// TwinCAT 3 PLC project Building_1_5_Totes_ARUP
// ProgramVersion: 3.1.4023.0
// libraries:
//   Tc2_Standard, * (Beckhoff Automation GmbH)
//   Tc2_System, * (Beckhoff Automation GmbH)
//   Tc2_TcpIp, * (Beckhoff Automation GmbH)
//   Tc2_Utilities, * (Beckhoff Automation GmbH)
//   Tc3_Module, * (Beckhoff Automation GmbH)
// project tree:
//   DUTs/EAP/ E_EAP_PubType.TcDUT, ST_EAP_DEVICE.TcDUT, ST_EAP_Publisher.TcDUT, ST_EAP_Pub_Variable.TcDUT, ST_EAP_Subscriber.TcDUT, ST_EAP_Sub_Variable.TcDUT
//   DUTs/ E_EquipType.TcTLEO, E_StatusCode.TcDUT, ST_EquipmentStatus.TcDUT, ST_SafetyState.TcDUT
//   DUTs/Messages/ E_EquipmentUpdate.TcTLEO, E_MessageIds.TcTLEO, E_TransportComplete.TcDUT, E_TransportResponse.TcTLEO, ST_Msg_ConveyorStat.TcDUT, ST_Msg_EquipStat.TcDUT
//   FunctionBlocks/BarCode/ CognexDataMan260.TcPOU
//   FunctionBlocks/Binder/ BinderX_ReleaseControl.TcPOU, FB_BinderPusher.TcPOU, FB_Binder_SingulateHold.TcPOU
//   FunctionBlocks/Binder/DUTs/ ST_Binder.TcDUT, ST_BinderState.TcDUT, ST_FromBinder.TcDUT, ST_ToBinder.TcDUT
//   FunctionBlocks/Conveyance/DUTs/ E_ConvType.TcDUT
//   FunctionBlocks/Conveyance/ FB_CnvyrCnfig_1.TcPOU, FB_SleepCntrl.TcPOU
//   FunctionBlocks/Divert/DUTs/ ST_Divert.TcDUT, ST_DivertCfg.TcDUT
//   FunctionBlocks/Divert/Functions/ FB_ConfirmCheck.TcPOU, FB_DivertCommission.TcPOU, FB_DivertControl.TcPOU, FB_DivertDecision.TcPOU, FB_DivertFullMonitor.TcPOU, FB_DivertLog.TcPOU
//   FunctionBlocks/Encoder/DUTs/ ST_Encoder.TcDUT
//   FunctionBlocks/Encoder/ FB_ProcessEncoder.TcPOU
//   FunctionBlocks/FB_Merge/ E_MergeState.TcDUT, FB_Merge2.TcPOU, MergeExample.TcPOU, ST_MergeSts.TcDUT
//   FunctionBlocks/FB_Merge/Merge Inlet/ FB_MergeInlet.TcPOU, ST_MergeInlet.TcDUT, ST_MergeInletCfg.TcDUT, ST_MergeInletCtrl.TcDUT, ST_MergeInletSts.TcDUT
//   FunctionBlocks/FB_MotionMerge/ FB_MotionMerge.TcPOU, MotionMergeExample.TcPOU, ST_MotionMergeConfig.TcDUT, ST_MotionMergeItem.TcDUT
//   FunctionBlocks/Item/DUTs/ ST_Item.TcDUT, ST_ItemBuffer.TcDUT, ST_ItemBufferFdbk.TcDUT, ST_ItemLogBuffer.TcDUT, ST_ItemTemporary.TcDUT
//   FunctionBlocks/Item/ FB_ItemBuffer.TcPOU, FB_ItemLogBuffer.TcPOU
//   FunctionBlocks/LEDControl/ FB_LEDModeCtrl.TcPOU, ST_HMILEDMode.TcDUT, ST_LEDMode.TcDUT, ST_RGB.TcDUT
//   FunctionBlocks/Logging/ FB_UpdateLog.TcPOU, ST_LogMsg.TcDUT
//   FunctionBlocks/Metrics/ FB_Metrics.TcPOU
//   FunctionBlocks/Server/Data types/ E_ConnectionSteps.TcDUT, E_ServerSteps.TcDUT
//   FunctionBlocks/Server/ FB_Server.TcPOU, FB_ServerApplication.TcPOU, FB_ServerConnection.TcPOU
//   FunctionBlocks/Server/Helper POUs/ FB_FrameFifo.TcPOU, FB_LogFifo.TcPOU
//   FunctionBlocks/Singulation/ FB_Singulation.TcPOU, FB_TwoGripIndexer.TcPOU, FB_TwoGripSingulation.TcPOU
//   FunctionBlocks/Solenoids/Functions/ FB_Solenoid_DA.TcPOU, FB_Solenoid_SA.TcPOU
//   FunctionBlocks/Sorter/DUTs/ ST_RoundRobin.TcDUT, ST_RoundRobinCfg.TcDUT, ST_RoundRobinDest.TcDUT, ST_Sorter.TcDUT, ST_SorterConfig.TcDUT
//   FunctionBlocks/Sorter/Functions/ FB_FindDestination.TcPOU, FB_SorterLog.TcPOU
//   FunctionBlocks/Sorter/ ProcessBuffers.TcPOU, SorterExample.TcPOU, SorterProgram.TcPOU
//   FunctionBlocks/Sorter/VISUs/ ArrayInspection.TcVIS, DiverterTest.TcVIS, SorterArray.TcVIS
//   FunctionBlocks/StateControl/ E_OperStateCntrl.TcTLEO, E_StateCntrl.TcTLEO, E_StopCodes.TcTLEO, FB_ManageCodes.TcPOU, FB_StateCntrl.TcPOU, ST_StateCntrlPB.TcDUT, ST_StateCntrlSts.TcDUT
//   FunctionBlocks/Utils/Events/ FB_EventMngr.TcPOU, FB_Intlks_Latch.TcPOU, FB_Intlks_NoLatch.TcPOU, ST_CfgEvents.TcDUT, ST_EventSts.TcDUT
//   FunctionBlocks/Utils/ FB_AlrtStrtDelay.TcPOU, FB_EquipCntrl.TcPOU, FB_Flasher.TcPOU, FB_FlipFlop.TcPOU, FB_JamDetect.TcPOU, FB_PhotoEye.TcPOU, FB_SystemCntrl.TcPOU, F_CalculateDifference.TcPOU, F_CalculateIndex.TcPOU, F_DecIndex.TcPOU, F_IncIndex.TcPOU, F_PaddNumber.TcPOU, IncIndex.TcPOU, SystemCntrl_Example.TcPOU
//   FunctionBlocks/Utils/Filters/ FB_DigDebnce.TcPOU, FB_DigDebnce_Off.TcPOU, FB_DigDebnce_On.TcPOU, F_Clip.TcPOU
//   FunctionBlocks/VFD/DUTs/ DRIVE_STATE.TcTLEO
//   FunctionBlocks/VFD/Functions/ DriveState.TcPOU, VFD.TcPOU
//   / GlobalTextList.TcGTLO, PlcTask.TcTTO, Visualization Manager.TcVMO (not stored)
//   GVLs/ GVL_EquipArrays.TcGVL, GVL_IO.TcGVL, GVL_Logging.TcGVL, GVL_SorterItems.TcGVL
//   POUs/ BarCodeReaders.TcPOU, CommStatus.TcPOU, Conveyors.TcPOU, Log_Diverts_P2140.TcPOU, Log_Diverts_P2150.TcPOU, MAIN.TcPOU, MsgControl.TcPOU, Photoeyes.TcPOU, ProcessBuffers_P2150.TcPOU, ProcessBuffers_P2140.TcPOU, ProxSensors.TcPOU, P_PulseCountDist.TcPOU, ServerControl.TcPOU, Singulation_Control.TcPOU, Solenoids.TcPOU, Sorter.TcPOU, Sorter_P2140.TcPOU, Sorter_P2150.TcPOU, System.TcPOU, SystemSafety.TcPOU
// real-time tasks:
//   TASK PlcTask: cycle T#10ms, priority 20, ADS port 350
//   TASK BCR_Sync: cycle T#1ms, priority 1, ADS port 301
// I/O:
//   DEVICE Device 1 (EtherCAT), AmsNetId 5.84.5.4.2.1
//     Term 1 (EK1200) [EK1200-5000 EtherCAT Power supply (2A E-Bus)]
//       Term 2 (EL6070-0033)
//       PLC-7021 (EL1008) [EL1008 8Ch. Dig. Input 24V, 3ms]
//       PLC-8051 (EL2008) [EL2008 8Ch. Dig. Output 24V, 0.5A]
//       PLC-8431 (EL1918) [EL1918, 8Ch. Safety Input 24V, TwinSAFE]
//         modules: Module 2 (FSLOGIC)
//       PLC-9031 (EL5152) [EL5152 2Ch. Inc. Encoder]
//       PLC-10081 (EK1122) [EK1122 2 port EtherCAT junction] // RIOs
//         SRIO-1151 (EP1908) [EP1908, 8 Ch. Safety Input 24V, TwinSAFE ]
//           modules: Module 1 (FSOE)
//         RIO-2151 (EP2339-0022) [EP2339-0022 16 Ch. Dig. Input/Output 24V, 0,5A, M12]
//         RIO-3171 (EP2339-0022) [EP2339-0022 16 Ch. Dig. Input/Output 24V, 0,5A, M12]
//         RIO-4141 (EP2339-0022) [EP2339-0022 16 Ch. Dig. Input/Output 24V, 0,5A, M12]
//         SRIO-7151 (EP1908) [EP1908, 8 Ch. Safety Input 24V, TwinSAFE ]
//           modules: Module 1 (FSOE)
//         RIO-8171 (EP2339-0022) [EP2339-0022 16 Ch. Dig. Input/Output 24V, 0,5A, M12]
//         RIO-9191 (EP2339-0022) [EP2339-0022 16 Ch. Dig. Input/Output 24V, 0,5A, M12]
//         RIO-10161 (EP2339-0022) [EP2339-0022 16 Ch. Dig. Input/Output 24V, 0,5A, M12]
//         RIO-11171 (EP2339-0022) [EP2339-0022 16 Ch. Dig. Input/Output 24V, 0,5A, M12]
//         RIO12182 (EP2339-0022) [EP2339-0022 16 Ch. Dig. Input/Output 24V, 0,5A, M12]
//       PLC-10261 (EK1122) [EK1122 2 port EtherCAT junction] // MCC
//         Term 19 (EK1100) [EK1100 EtherCAT Coupler (2A E-Bus)]
//           PLC-12031 (EL2008) [EL2008 8Ch. Dig. Output 24V, 0.5A]
//           PLC-12221 (EL2008) [EL2008 8Ch. Dig. Output 24V, 0.5A]
//           PLC-12451 (EL1008) [EL1008 8Ch. Dig. Input 24V, 3ms]
//           PLC-12631 (EL1008) [EL1008 8Ch. Dig. Input 24V, 3ms]
//           PLC-13071 (EL2008) [EL2008 8Ch. Dig. Output 24V, 0.5A]
//           PLC-13471 (EL1008) [EL1008 8Ch. Dig. Input 24V, 3ms]
//           PLC-14061 (EL1918) [EL1918, 8Ch. Safety Input 24V, TwinSAFE]
//             modules: Module 1 (FSOE), Module 2 (FSLOGIC)
//           PLC-14461 (EL2904) [EL2904, 4 Ch. Safety Output 24V, 0.5A, TwinSAFE]
//             modules: Module 1 (FSOES), Module 2 (DO)
//           PLC-15101 (EK1122) [EK1122 2 port EtherCAT junction]
//             P2141 (Inverter i550 Cabinet) [i550 Cabinet V05.04.xx]
//             P2146 (Inverter i550 Cabinet) [i550 Cabinet V06.02.xx]
//             P3080 (Inverter i550 Cabinet) [i550 Cabinet V06.02.xx]
//   DEVICE Device 2 (RT-Ethernet Protocol), AmsNetId 5.84.5.4.3.1
//   DEVICE Communition with 205 (EtherCAT Automation Protocol), AmsNetId 5.84.5.4.4.1
//     Pub_To_205 (Publisher)
//     Sub_To_205 (Subscriber)
//   DEVICE Device 4 (TC3 EIP Scanner), AmsNetId 5.84.5.2.5.1
//     BCR_S2140_01 // <INFO> </INFO> <EDS> C:\TwinCAT\3.1\Config\Io\EtherNetIP\0678077313070100.eds </EDS>
//     BCR_S2141_2 // <INFO> </INFO> <EDS> C:\TwinCAT\3.1\Config\Io\EtherNetIP\0678077313070100.eds </EDS>
//     BCR_S2150_2 // <INFO> </INFO> <EDS> C:\TwinCAT\3.1\Config\Io\EtherNetIP\0678077313070100.eds </EDS>
//     BCR_S3080_01 // <INFO> </INFO> <EDS> C:\TwinCAT\3.1\Config\Io\EtherNetIP\0678077313070100.eds </EDS>
// variable links:
//   (this object) <-> Device 1 (EtherCAT)/Term 1 (EK1200)/PLC-10081 (EK1122)/SRIO-1151 (EP1908)
//     Term 1 (EK1200)/PLC-8431 (EL1918)/ConnectionInputs/Message_26 TxPDO <-> Module 1 (FSOE)/FSOE Outputs/FSOE
//     Term 1 (EK1200)/PLC-8431 (EL1918)/ConnectionOutputs/Message_26 RxPDO <-> Module 1 (FSOE)/FSOE Inputs/FSOE
//   (this object) <-> Device 1 (EtherCAT)/Term 1 (EK1200)/PLC-10081 (EK1122)/SRIO-7151 (EP1908)
//     Term 1 (EK1200)/PLC-8431 (EL1918)/ConnectionInputs/Message_25 TxPDO <-> Module 1 (FSOE)/FSOE Outputs/FSOE
//     Term 1 (EK1200)/PLC-8431 (EL1918)/ConnectionOutputs/Message_25 RxPDO <-> Module 1 (FSOE)/FSOE Inputs/FSOE
//   (this object) <-> Device 1 (EtherCAT)/Term 1 (EK1200)/PLC-10261 (EK1122)/Term 19 (EK1100)/PLC-14061 (EL1918)
//     Term 1 (EK1200)/PLC-8431 (EL1918)/ConnectionInputs/Message_29 TxPDO <-> Module 1 (FSOE)/FSoE Outputs/FSOE
//     Term 1 (EK1200)/PLC-8431 (EL1918)/ConnectionOutputs/Message_29 RxPDO <-> Module 1 (FSOE)/FSoE Inputs/FSOE
//   (this object) <-> Device 1 (EtherCAT)/Term 1 (EK1200)/PLC-10261 (EK1122)/Term 19 (EK1100)/PLC-14461 (EL2904)
//     Term 1 (EK1200)/PLC-8431 (EL1918)/ConnectionInputs/Message_27 TxPDO <-> Module 1 (FSOES)/RxPDO/FSOE
//     Term 1 (EK1200)/PLC-8431 (EL1918)/ConnectionOutputs/Message_27 RxPDO <-> Module 1 (FSOES)/TxPDO/FSOE
//   (this object) <-> Device 1 (EtherCAT)/Term 1 (EK1200)/PLC-8431 (EL1918)
//     Term 1 (EK1200)/PLC-10081 (EK1122)/SRIO-1151 (EP1908)/Module 1 (FSOE)/FSOE Inputs/FSOE <-> ConnectionOutputs/Message_26 RxPDO
//     Term 1 (EK1200)/PLC-10081 (EK1122)/SRIO-7151 (EP1908)/Module 1 (FSOE)/FSOE Inputs/FSOE <-> ConnectionOutputs/Message_25 RxPDO
//     Term 1 (EK1200)/PLC-10081 (EK1122)/SRIO-1151 (EP1908)/Module 1 (FSOE)/FSOE Outputs/FSOE <-> ConnectionInputs/Message_26 TxPDO
//     Term 1 (EK1200)/PLC-10081 (EK1122)/SRIO-7151 (EP1908)/Module 1 (FSOE)/FSOE Outputs/FSOE <-> ConnectionInputs/Message_25 TxPDO
//     Term 1 (EK1200)/PLC-10261 (EK1122)/Term 19 (EK1100)/PLC-14061 (EL1918)/Module 1 (FSOE)/FSoE Inputs/FSOE <-> ConnectionOutputs/Message_29 RxPDO
//     Term 1 (EK1200)/PLC-10261 (EK1122)/Term 19 (EK1100)/PLC-14061 (EL1918)/Module 1 (FSOE)/FSoE Outputs/FSOE <-> ConnectionInputs/Message_29 TxPDO
//     Term 1 (EK1200)/PLC-10261 (EK1122)/Term 19 (EK1100)/PLC-14461 (EL2904)/Module 1 (FSOES)/RxPDO/FSOE <-> ConnectionInputs/Message_27 TxPDO
//     Term 1 (EK1200)/PLC-10261 (EK1122)/Term 19 (EK1100)/PLC-14461 (EL2904)/Module 1 (FSOES)/TxPDO/FSOE <-> ConnectionOutputs/Message_27 RxPDO
//   Building_1_5_Totes_ARUP Instance <-> Communition with 205 (EtherCAT Automation Protocol)
//     PlcTask Inputs/MAIN.EAP_205.DevState <-> Inputs/DevState
//     PlcTask Outputs/MAIN.EAP_205.DevCtrl <-> Outputs/DevCtrl
//   Building_1_5_Totes_ARUP Instance <-> Communition with 205 (EtherCAT Automation Protocol)/Pub_To_205 (Publisher)
//     PlcTask Inputs/MAIN.EAP_205.Publisher.FrameState <-> Inputs/FrameState
//     PlcTask Inputs/MAIN.EAP_205.Publisher.Variables[0].VarState <-> To205_P2130_IsRunning/Inputs/VarState
//     PlcTask Inputs/MAIN.EAP_205.Publisher.Variables[1].VarState <-> To205_P3095_SendingProduct/Inputs/VarState
//     PlcTask Outputs/GVL_IO.To205_P2130_IsRunning <-> To205_P2130_IsRunning/Outputs/VarData
//     PlcTask Outputs/GVL_IO.To205_P3095_SendingProduct <-> To205_P3095_SendingProduct/Outputs/VarData
//     PlcTask Outputs/MAIN.EAP_205.Publisher.FrameCtrl <-> Outputs/FrameCtrl
//     PlcTask Outputs/MAIN.EAP_205.Publisher.IPAddr <-> Outputs/IpAddr
//     PlcTask Outputs/MAIN.EAP_205.Publisher.Variables[0].VarCtrl <-> To205_P2130_IsRunning/Outputs/VarCtrl
//     PlcTask Outputs/MAIN.EAP_205.Publisher.Variables[0].VarID <-> To205_P2130_IsRunning/Outputs/VarId
//     PlcTask Outputs/MAIN.EAP_205.Publisher.Variables[1].VarCtrl <-> To205_P3095_SendingProduct/Outputs/VarCtrl
//     PlcTask Outputs/MAIN.EAP_205.Publisher.Variables[1].VarID <-> To205_P3095_SendingProduct/Outputs/VarId
//   Building_1_5_Totes_ARUP Instance <-> Communition with 205 (EtherCAT Automation Protocol)/Sub_To_205 (Subscriber)
//     PlcTask Inputs/GVL_IO.From205_P2125_SendingProduct <-> From205_P2125_SendingProduct/Inputs/VarData
//     PlcTask Inputs/GVL_IO.From205_P3100_IsRunning <-> From205_P3100_IsRunning/Inputs/VarData
//     PlcTask Inputs/MAIN.EAP_205.Subscriber.FrameState <-> Inputs/FrameState
//     PlcTask Inputs/MAIN.EAP_205.Subscriber.Variables[0].CycleIndex <-> From205_P3100_IsRunning/Inputs/CycleIndex
//     PlcTask Inputs/MAIN.EAP_205.Subscriber.Variables[0].Quality <-> From205_P3100_IsRunning/Inputs/Quality
//     PlcTask Inputs/MAIN.EAP_205.Subscriber.Variables[0].VarState <-> From205_P3100_IsRunning/Inputs/VarState
//     PlcTask Inputs/MAIN.EAP_205.Subscriber.Variables[1].CycleIndex <-> From205_P2125_SendingProduct/Inputs/CycleIndex
//     PlcTask Inputs/MAIN.EAP_205.Subscriber.Variables[1].Quality <-> From205_P2125_SendingProduct/Inputs/Quality
//     PlcTask Inputs/MAIN.EAP_205.Subscriber.Variables[1].VarState <-> From205_P2125_SendingProduct/Inputs/VarState
//     PlcTask Outputs/MAIN.EAP_205.Subscriber.FrameCtrl <-> Outputs/FrameCtrl
//     PlcTask Outputs/MAIN.EAP_205.Subscriber.Variables[0].VarCtrl <-> From205_P3100_IsRunning/Outputs/VarCtrl
//     PlcTask Outputs/MAIN.EAP_205.Subscriber.Variables[0].VarId <-> From205_P3100_IsRunning/Outputs/VarId
//     PlcTask Outputs/MAIN.EAP_205.Subscriber.Variables[1].VarCtrl <-> From205_P2125_SendingProduct/Outputs/VarCtrl
//     PlcTask Outputs/MAIN.EAP_205.Subscriber.Variables[1].VarId <-> From205_P2125_SendingProduct/Outputs/VarId
//   Building_1_5_Totes_ARUP Instance <-> Device 1 (EtherCAT)/Term 1 (EK1200)/PLC-10081 (EK1122)/RIO-10161 (EP2339-0022)
//     PlcTask Inputs/GVL_IO.DS_P2135 <-> Channel 8/P2135 Motor Disconnect
//     PlcTask Inputs/GVL_IO.DS_P2140 <-> Channel 2/P2140 Motor Disconnect
//     PlcTask Inputs/GVL_IO.PB_RemoteReset_10221 <-> Channel 6/PB-10221
//     PlcTask Inputs/Photoeyes.PE_10081.In_PE <-> Channel 9/PE-10081
//     PlcTask Inputs/Photoeyes.PE_10091.In_PE <-> Channel 1/PE-10091
//     PlcTask Inputs/Photoeyes.PE_10151.In_PE <-> Channel 11/PE-10151
//     PlcTask Inputs/Photoeyes.PE_10291.In_PE <-> Channel 7/PE-10291
//     PlcTask Inputs/Photoeyes.PE_10302.In_PE <-> Channel 15/PE-10302
//     PlcTask Inputs/ProxSensors.In_PX_10181_Extended <-> Channel 12/PX-10181
//     PlcTask Inputs/ProxSensors.In_PX_10211_Extended <-> Channel 13/PX-10211
//     PlcTask Inputs/ProxSensors.In_PX_10231_Retracted <-> Channel 14/PX-10231
//     PlcTask Outputs/GVL_IO.LT_10161_Red <-> Channel 19/LT-10161
//     PlcTask Outputs/GVL_IO.LT_10171_Yellow <-> Channel 20/LT-10171
//     PlcTask Outputs/GVL_IO.LT_10201_Green <-> Channel 21/LT-10201
//     PlcTask Outputs/GVL_IO.PL2140_01_Extend <-> Channel 26/SV-10121
//   Building_1_5_Totes_ARUP Instance <-> Device 1 (EtherCAT)/Term 1 (EK1200)/PLC-10081 (EK1122)/RIO-11171 (EP2339-0022)
//     PlcTask Inputs/GVL_IO.RIO11171_WcState <-> WcState/WcState
//     PlcTask Inputs/Photoeyes.PE_11191.In_PE <-> Channel 11/PE-11191
//     PlcTask Inputs/Photoeyes.PE_11221.In_PE <-> Channel 12/PE11221
//     PlcTask Inputs/Photoeyes.PE_11241.In_PE <-> Channel 13/????PE11421
//     PlcTask Inputs/ProxSensors.In_PX_11141_Extended <-> Channel 9/PX-11141
//     PlcTask Inputs/ProxSensors.In_PX_11181_Extended <-> Channel 3/PX-11181
//     PlcTask Inputs/ProxSensors.In_PX_11291_Extended <-> Channel 7/PX-11291
//     PlcTask Inputs/ProxSensors.In_PX_11161_Retracted <-> Channel 10/PX-11161
//     PlcTask Inputs/ProxSensors.In_PX_11201_Retracted <-> Channel 4/PX-11201
//     PlcTask Inputs/ProxSensors.In_PX_11321_Retracted <-> Channel 8/PX-11321
//     PlcTask Outputs/GVL_IO.GR2140_01_Extend <-> Channel 22/SV-11261
//     PlcTask Outputs/GVL_IO.GR2140_02_Extend <-> Channel 21/SV-11241
//     PlcTask Outputs/GVL_IO.PI2140_01_Extend <-> Channel 17/SV-11121
//     PlcTask Outputs/GVL_IO.PI2140_01_Retract <-> Channel 18/SV-11151
//   Building_1_5_Totes_ARUP Instance <-> Device 1 (EtherCAT)/Term 1 (EK1200)/PLC-10081 (EK1122)/RIO-2151 (EP2339-0022)
//     PlcTask Inputs/GVL_IO.DS_P2145 <-> Channel 15/P2145 Motor Disconnect
//     PlcTask Inputs/GVL_IO.DS_P2146 <-> Channel 12/P2146 Motor Disconnect
//     PlcTask Inputs/GVL_IO.RIO2151_WcState <-> WcState/WcState
//     PlcTask Inputs/Photoeyes.PE_2101.In_PE <-> Channel 9/PE-2101
//     PlcTask Inputs/Photoeyes.PE_2131.In_PE <-> Channel 11/PE-2131
//     PlcTask Inputs/Photoeyes.PE_2201.In_PE <-> Channel 13/PE-2201
//     PlcTask Inputs/Photoeyes.PE_2231.In_PE <-> Channel 14/PE-2231
//     PlcTask Inputs/Photoeyes.PE_2301.In_PE <-> Channel 7/PE-2301
//     PlcTask Inputs/Photoeyes.PE_2331.In_PE <-> Channel 8/PE-2331
//     PlcTask Inputs/ProxSensors.In_PX_2131_Extended <-> Channel 1/PX-2131
//     PlcTask Inputs/ProxSensors.In_PX_2181_Extended <-> Channel 3/PX-2181
//     PlcTask Inputs/ProxSensors.In_PX_2151_Retracted <-> Channel 2/PX-2151
//     PlcTask Inputs/ProxSensors.In_PX_2201_Retracted <-> Channel 4/PX-2201
//     PlcTask Outputs/GVL_IO.GR2150_01_Extend <-> Channel 22/SV-2261
//     PlcTask Outputs/GVL_IO.PI2150_01_Extend <-> Channel 21/SV-2241
//   Building_1_5_Totes_ARUP Instance <-> Device 1 (EtherCAT)/Term 1 (EK1200)/PLC-10081 (EK1122)/RIO-3171 (EP2339-0022)
//     PlcTask Inputs/GVL_IO.PB_RemoteReset_3211 <-> Channel 12/PB-3211
//     PlcTask Inputs/GVL_IO.RIO3171_WcState <-> WcState/WcState
//     PlcTask Inputs/Photoeyes.PE_3111.In_PE <-> Channel 1/PE-3111
//     PlcTask Inputs/Photoeyes.PE_3231.In_PE <-> Channel 5/PE-3231
//     PlcTask Inputs/ProxSensors.In_PX_3171_Extended <-> Channel 3/PX-3171
//     PlcTask Inputs/ProxSensors.In_PX_3301_Extended <-> Channel 7/PX-3301
//     PlcTask Inputs/ProxSensors.In_PX_3191_Retracted <-> Channel 4/PX-3191
//     PlcTask Inputs/ProxSensors.In_PX_3331_Retracted <-> Channel 8/PX-3331
//     PlcTask Outputs/GVL_IO.LT_3131_Red <-> Channel 25/LT-3131
//     PlcTask Outputs/GVL_IO.LT_3151_Yellow <-> Channel 26/LT-3151
//     PlcTask Outputs/GVL_IO.LT_3201_Green <-> Channel 27/LT-3201
//     PlcTask Outputs/GVL_IO.PU2150_01_Extend <-> Channel 22/SV-3261
//     PlcTask Outputs/GVL_IO.PU2150_02_Extend <-> Channel 18/SV-3141
//   Building_1_5_Totes_ARUP Instance <-> Device 1 (EtherCAT)/Term 1 (EK1200)/PLC-10081 (EK1122)/RIO-4141 (EP2339-0022)
//     PlcTask Inputs/GVL_IO.DS_P2150 <-> Channel 9/P2150 Motor Discconnect
//     PlcTask Inputs/GVL_IO.RIO4141_WcState <-> WcState/WcState
//     PlcTask Inputs/Photoeyes.PE_4091.In_PE <-> Channel 1/PE-4091
//     PlcTask Inputs/Photoeyes.PE_4161.In_PE <-> Channel 11/PE-4161
//     PlcTask Inputs/Photoeyes.PE_4201.In_PE <-> Channel 5/PE-4201
//     PlcTask Inputs/ProxSensors.In_PX_4151_Extended <-> Channel 3/PX-4151
//     PlcTask Inputs/ProxSensors.In_PX_4291_Extended <-> Channel 7/PX-4291
//     PlcTask Inputs/ProxSensors.In_PX_4171_Retracted <-> Channel 4/PX-4171
//     PlcTask Inputs/ProxSensors.In_PX_4311_Retracted <-> Channel 8/PX-4311
//     PlcTask Outputs/GVL_IO.PU2150_03_Extend <-> Channel 22/SV-4241
//     PlcTask Outputs/GVL_IO.PU2150_04_Extend <-> Channel 18/SV-4121
//   Building_1_5_Totes_ARUP Instance <-> Device 1 (EtherCAT)/Term 1 (EK1200)/PLC-10081 (EK1122)/RIO-8171 (EP2339-0022)
//     PlcTask Inputs/GVL_IO.DS_P2141 <-> Channel 7/P2141 Motor Disconnect
//     PlcTask Inputs/GVL_IO.DS_P2142 <-> Channel 1/P2142 Motor Disconnect
//     PlcTask Inputs/GVL_IO.DS_P2143 <-> Channel 8/P2143 Motor Disconnect
//     PlcTask Inputs/GVL_IO.PB_RemoteReset_8251 <-> Channel 6/PB-8251
//     PlcTask Inputs/GVL_IO.RIO8171_WcState <-> WcState/WcState
//     PlcTask Inputs/Photoeyes.PE_8131.In_PE <-> Channel 9/PE-8131
//     PlcTask Inputs/Photoeyes.PE_8141.In_PE <-> Channel 2/PE-8141
//     PlcTask Inputs/Photoeyes.PE_8161.In_PE <-> Channel 10/PE-8161
//     PlcTask Outputs/GVL_IO.LT_8181_Red <-> Channel 19/LT-8181
//     PlcTask Outputs/GVL_IO.LT_8191_Yellow <-> Channel 20/LT-8191
//     PlcTask Outputs/GVL_IO.LT_8231_Green <-> Channel 21/LT-8231
//   Building_1_5_Totes_ARUP Instance <-> Device 1 (EtherCAT)/Term 1 (EK1200)/PLC-10081 (EK1122)/RIO-9191 (EP2339-0022)
//     PlcTask Inputs/GVL_IO.DS_P3080 <-> Channel 5/P3080 Motor Disconnect
//     PlcTask Inputs/GVL_IO.RIO9191_WcState <-> WcState/WcState
//     PlcTask Inputs/Photoeyes.PE_9141.In_PE <-> Channel 1/PE-9141
//     PlcTask Inputs/Photoeyes.PE_9161.In_PE <-> Channel 2/PE-9161
//     PlcTask Inputs/Photoeyes.PE_9191.In_PE <-> Channel 3/PE-9191
//     PlcTask Inputs/Photoeyes.PE_9221.In_PE <-> Channel 4/PE-9221
//   Building_1_5_Totes_ARUP Instance <-> Device 1 (EtherCAT)/Term 1 (EK1200)/PLC-10081 (EK1122)/RIO12182 (EP2339-0022)
//     PlcTask Inputs/GVL_IO.DS_P2130 <-> Channel 4/P2130 Motor Disconnect
//     PlcTask Inputs/GVL_IO.DS_P3085 <-> Channel 2/P3085 Motor Disconnect
//     PlcTask Inputs/GVL_IO.DS_P3090 <-> Channel 6/P3090 Motor Disconnect
//     PlcTask Inputs/GVL_IO.DS_P3095 <-> Channel 12/P3095 Motor Disconnect
//     PlcTask Inputs/GVL_IO.RIO12182_WcState <-> WcState/WcState
//     PlcTask Inputs/Photoeyes.PE_12091.In_PE <-> Channel 1/PE-12091
//     PlcTask Inputs/Photoeyes.PE_12121.In_PE <-> Channel 9/PE-12121
//     PlcTask Inputs/Photoeyes.PE_12171.In_PE <-> Channel 3/PE-12171
//     PlcTask Inputs/Photoeyes.PE_12181.In_PE <-> Channel 11/PE-12181
//     PlcTask Inputs/Photoeyes.PE_12271.In_PE <-> Channel 5/PE-12271
//     PlcTask Inputs/ProxSensors.In_PX_12151_Extended <-> Channel 10/PX-12151
//     PlcTask Inputs/ProxSensors.In_PX_12251_Extended <-> Channel 13/PX-12251
//   Building_1_5_Totes_ARUP Instance <-> Device 1 (EtherCAT)/Term 1 (EK1200)/PLC-10081 (EK1122)/SRIO-1151 (EP1908)
//     PlcTask Inputs/GVL_IO.RIO1151_WcState <-> WcState/WcState
//   Building_1_5_Totes_ARUP Instance <-> Device 1 (EtherCAT)/Term 1 (EK1200)/PLC-10081 (EK1122)/SRIO-7151 (EP1908)
//     PlcTask Inputs/GVL_IO.RIO7151_WcState <-> WcState/WcState
//   Building_1_5_Totes_ARUP Instance <-> Device 1 (EtherCAT)/Term 1 (EK1200)/PLC-10261 (EK1122)/Term 19 (EK1100)/PLC-12031 (EL2008)
//     PlcTask Outputs/GVL_IO.P2130_RUN <-> Channel 1/P2130 Run
//     PlcTask Outputs/GVL_IO.P2135_RUN <-> Channel 2/P2135 Run
//     PlcTask Outputs/GVL_IO.P2140_RUN <-> Channel 3/P2140 Run
//     PlcTask Outputs/GVL_IO.P2142_RUN <-> Channel 4/P2142 Run
//     PlcTask Outputs/GVL_IO.P2143_RUN <-> Channel 5/P2143 Run
//     PlcTask Outputs/GVL_IO.P2145_RUN <-> Channel 6/P2145 Run
//     PlcTask Outputs/GVL_IO.P2150_RUN <-> Channel 7/P2150 Run
//     PlcTask Outputs/GVL_IO.P3085_RUN <-> Channel 8/P3085 Run
//   Building_1_5_Totes_ARUP Instance <-> Device 1 (EtherCAT)/Term 1 (EK1200)/PLC-10261 (EK1122)/Term 19 (EK1100)/PLC-12221 (EL2008)
//     PlcTask Outputs/GVL_IO.P3090_RUN <-> Channel 1/P3090 Run
//     PlcTask Outputs/GVL_IO.P3095_RUN <-> Channel 2/P3095 Run
//   Building_1_5_Totes_ARUP Instance <-> Device 1 (EtherCAT)/Term 1 (EK1200)/PLC-10261 (EK1122)/Term 19 (EK1100)/PLC-12451 (EL1008)
//     PlcTask Inputs/GVL_IO.P2130_Faulted <-> Channel 1/P2130 Faulted
//     PlcTask Inputs/GVL_IO.P2135_Faulted <-> Channel 2/P2135 Faulted
//     PlcTask Inputs/GVL_IO.P2140_Faulted <-> Channel 3/P2140 Faulted
//     PlcTask Inputs/GVL_IO.P2142_Faulted <-> Channel 4/P2142 Faulted
//     PlcTask Inputs/GVL_IO.P2143_Faulted <-> Channel 5/P2143 Faulted
//     PlcTask Inputs/GVL_IO.P2145_Faulted <-> Channel 6/P2145 Faulted
//     PlcTask Inputs/GVL_IO.P2150_Faulted <-> Channel 7/P2150 Faulted
//     PlcTask Inputs/GVL_IO.P3085_Faulted <-> Channel 8/P3085 Faulted
//   Building_1_5_Totes_ARUP Instance <-> Device 1 (EtherCAT)/Term 1 (EK1200)/PLC-10261 (EK1122)/Term 19 (EK1100)/PLC-12631 (EL1008)
//     PlcTask Inputs/GVL_IO.P3090_Faulted <-> Channel 1/P3090 Faulted
//     PlcTask Inputs/GVL_IO.P3095_Faulted <-> Channel 2/P3095 Faulted
//   Building_1_5_Totes_ARUP Instance <-> Device 1 (EtherCAT)/Term 1 (EK1200)/PLC-10261 (EK1122)/Term 19 (EK1100)/PLC-15101 (EK1122)/P2141 (Inverter i550 Cabinet)
//     PlcTask Inputs/Conveyors.P2141_VFD.ActualVelocity <-> TPDO (A) Velocity/Actual speed
//     PlcTask Inputs/Conveyors.P2141_VFD.StatusWord <-> TPDO (A) Velocity/CiA status word
//     PlcTask Outputs/Conveyors.P2141_VFD.ControlWord <-> RPDO (A) Velocity/CiA control word
//     PlcTask Outputs/Conveyors.P2141_VFD.TargetVelocity <-> RPDO (A) Velocity/Set speed
//   Building_1_5_Totes_ARUP Instance <-> Device 1 (EtherCAT)/Term 1 (EK1200)/PLC-10261 (EK1122)/Term 19 (EK1100)/PLC-15101 (EK1122)/P2146 (Inverter i550 Cabinet)
//     PlcTask Inputs/Conveyors.P2146_VFD.ActualVelocity <-> TPDO (A) Velocity/Actual speed
//     PlcTask Inputs/Conveyors.P2146_VFD.StatusWord <-> TPDO (A) Velocity/CiA status word
//     PlcTask Outputs/Conveyors.P2146_VFD.ControlWord <-> RPDO (A) Velocity/CiA control word
//     PlcTask Outputs/Conveyors.P2146_VFD.TargetVelocity <-> RPDO (A) Velocity/Set speed
//   Building_1_5_Totes_ARUP Instance <-> Device 1 (EtherCAT)/Term 1 (EK1200)/PLC-10261 (EK1122)/Term 19 (EK1100)/PLC-15101 (EK1122)/P3080 (Inverter i550 Cabinet)
//     PlcTask Inputs/Conveyors.P3080_VFD.ActualVelocity <-> TPDO (A) Velocity/Actual speed
//     PlcTask Inputs/Conveyors.P3080_VFD.StatusWord <-> TPDO (A) Velocity/CiA status word
//     PlcTask Outputs/Conveyors.P3080_VFD.ControlWord <-> RPDO (A) Velocity/CiA control word
//     PlcTask Outputs/Conveyors.P3080_VFD.TargetVelocity <-> RPDO (A) Velocity/Set speed
//   Building_1_5_Totes_ARUP Instance <-> Device 1 (EtherCAT)/Term 1 (EK1200)/PLC-7021 (EL1008)
//     PlcTask Inputs/GVL_IO.PB_SysReset <-> Channel 3/PB-7061
//     PlcTask Inputs/GVL_IO.PB_SysStart <-> Channel 1/PB-7021
//     PlcTask Inputs/GVL_IO.PB_SysStop <-> Channel 2/PB-7041
//   Building_1_5_Totes_ARUP Instance <-> Device 1 (EtherCAT)/Term 1 (EK1200)/PLC-8051 (EL2008)
//     PlcTask Outputs/GVL_IO.HornMainPanel <-> Channel 1/AH-8051
//     PlcTask Outputs/GVL_IO.LT_MainPanelStack_Green <-> Channel 4/LT-8111
//     PlcTask Outputs/GVL_IO.LT_MainPanelStack_Red <-> Channel 2/LT-8071
//     PlcTask Outputs/GVL_IO.LT_MainPanelStack_Yellow <-> Channel 3/LT-8091
//   Building_1_5_Totes_ARUP Instance <-> Device 1 (EtherCAT)/Term 1 (EK1200)/PLC-8431 (EL1918)
//     PlcTask Inputs/GVL_IO.Remote_PullCord2142_OK <-> StandardInputs/Standard Out Var 10
//     PlcTask Inputs/GVL_IO.Remote_PullCord2150_OK <-> StandardInputs/Standard Out Var 28
//     PlcTask Inputs/SystemSafety.Safety_PanelEstop <-> StandardInputs/Standard Out Var 9
//     PlcTask Inputs/SystemSafety.Safety_SystemEstopsOK <-> StandardInputs/Standard Out Var 15
//     PlcTask Inputs/SystemSafety.System_SafetyState.ComErr <-> StandardInputs/Standard Out Var 16
//     PlcTask Inputs/SystemSafety.System_SafetyState.FBErr <-> StandardInputs/Standard Out Var 17
//     PlcTask Inputs/SystemSafety.System_SafetyState.InRun <-> StandardInputs/Standard Out Var 30
//     PlcTask Inputs/SystemSafety.System_SafetyState.OtherErr <-> StandardInputs/Standard Out Var 18
//     PlcTask Outputs/SystemSafety.System_SafetyState.CommErrAck <-> StandardOutputs/Standard In Var 31
//     PlcTask Outputs/SystemSafety.System_SafetyState.ErrAck <-> StandardOutputs/Standard In Var 1
//     PlcTask Outputs/SystemSafety.System_SafetyState.Reset <-> StandardOutputs/Standard In Var 5
//     PlcTask Outputs/SystemSafety.System_SafetyState.Run <-> StandardOutputs/Standard In Var 2
//   Building_1_5_Totes_ARUP Instance <-> Device 1 (EtherCAT)/Term 1 (EK1200)/PLC-9031 (EL5152)
//     PlcTask Inputs/GVL_IO.ENC_9031_Period <-> ENC Period Channel 2/Period value
//     PlcTask Inputs/GVL_IO.ENC_9091_Period <-> ENC Period Channel 1/Period value
//     PlcTask Inputs/GVL_IO.ENC_9031_Raw <-> ENC Status compact Channel 2/Counter value
//     PlcTask Inputs/GVL_IO.ENC_9091_Raw <-> ENC Status compact Channel 1/Counter value
//   Building_1_5_Totes_ARUP Instance <-> Device 2 (RT-Ethernet Protocol)
//     PlcTask Inputs/GVL_IO.EthernetAdapter_State <-> Inputs/DevState
//   Building_1_5_Totes_ARUP Instance <-> Device 4 (TC3 EIP Scanner)/BCR_S2140_01
//     PlcTask Inputs/BarCodeReaders.BCR_S2140_01.Acquiring <-> Connection 1 (Input/Output)/Inputs/Acquiring
//     PlcTask Inputs/BarCodeReaders.BCR_S2140_01.DecodeComplete <-> Connection 1 (Input/Output)/Inputs/Decode Complete
//     PlcTask Inputs/BarCodeReaders.BCR_S2140_01.Decoding <-> Connection 1 (Input/Output)/Inputs/Decoding
//     PlcTask Inputs/BarCodeReaders.BCR_S2140_01.DeviceState <-> Inputs/State
//     PlcTask Inputs/BarCodeReaders.BCR_S2140_01.ResultCode <-> Connection 1 (Input/Output)/Inputs/Result Code
//     PlcTask Inputs/BarCodeReaders.BCR_S2140_01.ResultData <-> Connection 1 (Input/Output)/Inputs/Result Data
//     PlcTask Inputs/BarCodeReaders.BCR_S2140_01.ResultData @bit 8 <-> Connection 1 (Input/Output)/Inputs/Result Data_1
//     PlcTask Inputs/BarCodeReaders.BCR_S2140_01.ResultData @bit 80 <-> Connection 1 (Input/Output)/Inputs/Result Data_10
//     PlcTask Inputs/BarCodeReaders.BCR_S2140_01.ResultData @bit 88 <-> Connection 1 (Input/Output)/Inputs/Result Data_11
//     PlcTask Inputs/BarCodeReaders.BCR_S2140_01.ResultData @bit 96 <-> Connection 1 (Input/Output)/Inputs/Result Data_12
//     PlcTask Inputs/BarCodeReaders.BCR_S2140_01.ResultData @bit 104 <-> Connection 1 (Input/Output)/Inputs/Result Data_13
//     PlcTask Inputs/BarCodeReaders.BCR_S2140_01.ResultData @bit 112 <-> Connection 1 (Input/Output)/Inputs/Result Data_14
//     PlcTask Inputs/BarCodeReaders.BCR_S2140_01.ResultData @bit 120 <-> Connection 1 (Input/Output)/Inputs/Result Data_15
//     PlcTask Inputs/BarCodeReaders.BCR_S2140_01.ResultData @bit 128 <-> Connection 1 (Input/Output)/Inputs/Result Data_16
//     PlcTask Inputs/BarCodeReaders.BCR_S2140_01.ResultData @bit 136 <-> Connection 1 (Input/Output)/Inputs/Result Data_17
//     PlcTask Inputs/BarCodeReaders.BCR_S2140_01.ResultData @bit 144 <-> Connection 1 (Input/Output)/Inputs/Result Data_18
//     PlcTask Inputs/BarCodeReaders.BCR_S2140_01.ResultData @bit 152 <-> Connection 1 (Input/Output)/Inputs/Result Data_19
//     PlcTask Inputs/BarCodeReaders.BCR_S2140_01.ResultData @bit 16 <-> Connection 1 (Input/Output)/Inputs/Result Data_2
//     PlcTask Inputs/BarCodeReaders.BCR_S2140_01.ResultData @bit 160 <-> Connection 1 (Input/Output)/Inputs/Result Data_20
//     PlcTask Inputs/BarCodeReaders.BCR_S2140_01.ResultData @bit 168 <-> Connection 1 (Input/Output)/Inputs/Result Data_21
//     PlcTask Inputs/BarCodeReaders.BCR_S2140_01.ResultData @bit 176 <-> Connection 1 (Input/Output)/Inputs/Result Data_22
//     PlcTask Inputs/BarCodeReaders.BCR_S2140_01.ResultData @bit 184 <-> Connection 1 (Input/Output)/Inputs/Result Data_23
//     PlcTask Inputs/BarCodeReaders.BCR_S2140_01.ResultData @bit 192 <-> Connection 1 (Input/Output)/Inputs/Result Data_24
//     PlcTask Inputs/BarCodeReaders.BCR_S2140_01.ResultData @bit 200 <-> Connection 1 (Input/Output)/Inputs/Result Data_25
//     PlcTask Inputs/BarCodeReaders.BCR_S2140_01.ResultData @bit 24 <-> Connection 1 (Input/Output)/Inputs/Result Data_3
//     PlcTask Inputs/BarCodeReaders.BCR_S2140_01.ResultData @bit 32 <-> Connection 1 (Input/Output)/Inputs/Result Data_4
//     PlcTask Inputs/BarCodeReaders.BCR_S2140_01.ResultData @bit 40 <-> Connection 1 (Input/Output)/Inputs/Result Data_5
//     PlcTask Inputs/BarCodeReaders.BCR_S2140_01.ResultData @bit 48 <-> Connection 1 (Input/Output)/Inputs/Result Data_6
//     PlcTask Inputs/BarCodeReaders.BCR_S2140_01.ResultData @bit 56 <-> Connection 1 (Input/Output)/Inputs/Result Data_7
//     PlcTask Inputs/BarCodeReaders.BCR_S2140_01.ResultData @bit 64 <-> Connection 1 (Input/Output)/Inputs/Result Data_8
//     PlcTask Inputs/BarCodeReaders.BCR_S2140_01.ResultData @bit 72 <-> Connection 1 (Input/Output)/Inputs/Result Data_9
//     PlcTask Inputs/BarCodeReaders.BCR_S2140_01.ResultID <-> Connection 1 (Input/Output)/Inputs/Result ID
//     PlcTask Inputs/BarCodeReaders.BCR_S2140_01.ResultLength <-> Connection 1 (Input/Output)/Inputs/Result Length
//     PlcTask Inputs/BarCodeReaders.BCR_S2140_01.ResultsAvail <-> Connection 1 (Input/Output)/Inputs/Results Available
//     PlcTask Inputs/BarCodeReaders.BCR_S2140_01.TriggerAck <-> Connection 1 (Input/Output)/Inputs/Trigger Ack
//     PlcTask Inputs/BarCodeReaders.BCR_S2140_01.TriggerID <-> Connection 1 (Input/Output)/Inputs/Trigger ID
//     PlcTask Inputs/BarCodeReaders.BCR_S2140_01.TriggerReady <-> Connection 1 (Input/Output)/Inputs/Trigger Ready
//     PlcTask Outputs/BarCodeReaders.BCR_S2140_01.ResultsAck <-> Connection 1 (Input/Output)/Outputs/Results Ack
//     PlcTask Outputs/BarCodeReaders.BCR_S2140_01.Trigger <-> Connection 1 (Input/Output)/Outputs/Trigger
//     PlcTask Outputs/BarCodeReaders.BCR_S2140_01.TriggerEnable <-> Connection 1 (Input/Output)/Outputs/Trigger Enable
//   Building_1_5_Totes_ARUP Instance <-> Device 4 (TC3 EIP Scanner)/BCR_S2141_2
//     PlcTask Inputs/BarCodeReaders.BCR_S2141_01.Acquiring <-> Connection 2 (Input/Output)/Inputs/Acquiring
//     PlcTask Inputs/BarCodeReaders.BCR_S2141_01.DecodeComplete <-> Connection 2 (Input/Output)/Inputs/Decode Complete
//     PlcTask Inputs/BarCodeReaders.BCR_S2141_01.Decoding <-> Connection 2 (Input/Output)/Inputs/Decoding
//     PlcTask Inputs/BarCodeReaders.BCR_S2141_01.DeviceState <-> Inputs/State
//     PlcTask Inputs/BarCodeReaders.BCR_S2141_01.ResultCode <-> Connection 2 (Input/Output)/Inputs/Result Code
//     PlcTask Inputs/BarCodeReaders.BCR_S2141_01.ResultData <-> Connection 2 (Input/Output)/Inputs/Result Data
//     PlcTask Inputs/BarCodeReaders.BCR_S2141_01.ResultData @bit 8 <-> Connection 2 (Input/Output)/Inputs/Result Data_1
//     PlcTask Inputs/BarCodeReaders.BCR_S2141_01.ResultData @bit 80 <-> Connection 2 (Input/Output)/Inputs/Result Data_10
//     PlcTask Inputs/BarCodeReaders.BCR_S2141_01.ResultData @bit 88 <-> Connection 2 (Input/Output)/Inputs/Result Data_11
//     PlcTask Inputs/BarCodeReaders.BCR_S2141_01.ResultData @bit 96 <-> Connection 2 (Input/Output)/Inputs/Result Data_12
//     PlcTask Inputs/BarCodeReaders.BCR_S2141_01.ResultData @bit 104 <-> Connection 2 (Input/Output)/Inputs/Result Data_13
//     PlcTask Inputs/BarCodeReaders.BCR_S2141_01.ResultData @bit 112 <-> Connection 2 (Input/Output)/Inputs/Result Data_14
//     PlcTask Inputs/BarCodeReaders.BCR_S2141_01.ResultData @bit 120 <-> Connection 2 (Input/Output)/Inputs/Result Data_15
//     PlcTask Inputs/BarCodeReaders.BCR_S2141_01.ResultData @bit 128 <-> Connection 2 (Input/Output)/Inputs/Result Data_16
//     PlcTask Inputs/BarCodeReaders.BCR_S2141_01.ResultData @bit 136 <-> Connection 2 (Input/Output)/Inputs/Result Data_17
//     PlcTask Inputs/BarCodeReaders.BCR_S2141_01.ResultData @bit 144 <-> Connection 2 (Input/Output)/Inputs/Result Data_18
//     PlcTask Inputs/BarCodeReaders.BCR_S2141_01.ResultData @bit 152 <-> Connection 2 (Input/Output)/Inputs/Result Data_19
//     PlcTask Inputs/BarCodeReaders.BCR_S2141_01.ResultData @bit 16 <-> Connection 2 (Input/Output)/Inputs/Result Data_2
//     PlcTask Inputs/BarCodeReaders.BCR_S2141_01.ResultData @bit 160 <-> Connection 2 (Input/Output)/Inputs/Result Data_20
//     PlcTask Inputs/BarCodeReaders.BCR_S2141_01.ResultData @bit 168 <-> Connection 2 (Input/Output)/Inputs/Result Data_21
//     PlcTask Inputs/BarCodeReaders.BCR_S2141_01.ResultData @bit 176 <-> Connection 2 (Input/Output)/Inputs/Result Data_22
//     PlcTask Inputs/BarCodeReaders.BCR_S2141_01.ResultData @bit 184 <-> Connection 2 (Input/Output)/Inputs/Result Data_23
//     PlcTask Inputs/BarCodeReaders.BCR_S2141_01.ResultData @bit 192 <-> Connection 2 (Input/Output)/Inputs/Result Data_24
//     PlcTask Inputs/BarCodeReaders.BCR_S2141_01.ResultData @bit 200 <-> Connection 2 (Input/Output)/Inputs/Result Data_25
//     PlcTask Inputs/BarCodeReaders.BCR_S2141_01.ResultData @bit 24 <-> Connection 2 (Input/Output)/Inputs/Result Data_3
//     PlcTask Inputs/BarCodeReaders.BCR_S2141_01.ResultData @bit 32 <-> Connection 2 (Input/Output)/Inputs/Result Data_4
//     PlcTask Inputs/BarCodeReaders.BCR_S2141_01.ResultData @bit 40 <-> Connection 2 (Input/Output)/Inputs/Result Data_5
//     PlcTask Inputs/BarCodeReaders.BCR_S2141_01.ResultData @bit 48 <-> Connection 2 (Input/Output)/Inputs/Result Data_6
//     PlcTask Inputs/BarCodeReaders.BCR_S2141_01.ResultData @bit 56 <-> Connection 2 (Input/Output)/Inputs/Result Data_7
//     PlcTask Inputs/BarCodeReaders.BCR_S2141_01.ResultData @bit 64 <-> Connection 2 (Input/Output)/Inputs/Result Data_8
//     PlcTask Inputs/BarCodeReaders.BCR_S2141_01.ResultData @bit 72 <-> Connection 2 (Input/Output)/Inputs/Result Data_9
//     PlcTask Inputs/BarCodeReaders.BCR_S2141_01.ResultID <-> Connection 2 (Input/Output)/Inputs/Result ID
//     PlcTask Inputs/BarCodeReaders.BCR_S2141_01.ResultLength <-> Connection 2 (Input/Output)/Inputs/Result Length
//     PlcTask Inputs/BarCodeReaders.BCR_S2141_01.ResultsAvail <-> Connection 2 (Input/Output)/Inputs/Results Available
//     PlcTask Inputs/BarCodeReaders.BCR_S2141_01.TriggerAck <-> Connection 2 (Input/Output)/Inputs/Trigger Ack
//     PlcTask Inputs/BarCodeReaders.BCR_S2141_01.TriggerID <-> Connection 2 (Input/Output)/Inputs/Trigger ID
//     PlcTask Inputs/BarCodeReaders.BCR_S2141_01.TriggerReady <-> Connection 2 (Input/Output)/Inputs/Trigger Ready
//     PlcTask Outputs/BarCodeReaders.BCR_S2141_01.ResultsAck <-> Connection 2 (Input/Output)/Outputs/Results Ack
//     PlcTask Outputs/BarCodeReaders.BCR_S2141_01.Trigger <-> Connection 2 (Input/Output)/Outputs/Trigger
//     PlcTask Outputs/BarCodeReaders.BCR_S2141_01.TriggerEnable <-> Connection 2 (Input/Output)/Outputs/Trigger Enable
//   Building_1_5_Totes_ARUP Instance <-> Device 4 (TC3 EIP Scanner)/BCR_S2150_2
//     PlcTask Inputs/BarCodeReaders.BCR_S2150_01.Acquiring <-> Connection 2 (Input/Output)/Inputs/Acquiring
//     PlcTask Inputs/BarCodeReaders.BCR_S2150_01.DecodeComplete <-> Connection 2 (Input/Output)/Inputs/Decode Complete
//     PlcTask Inputs/BarCodeReaders.BCR_S2150_01.Decoding <-> Connection 2 (Input/Output)/Inputs/Decoding
//     PlcTask Inputs/BarCodeReaders.BCR_S2150_01.DeviceState <-> Inputs/State
//     PlcTask Inputs/BarCodeReaders.BCR_S2150_01.ResultCode <-> Connection 2 (Input/Output)/Inputs/Result Code
//     PlcTask Inputs/BarCodeReaders.BCR_S2150_01.ResultData <-> Connection 2 (Input/Output)/Inputs/Result Data
//     PlcTask Inputs/BarCodeReaders.BCR_S2150_01.ResultData @bit 8 <-> Connection 2 (Input/Output)/Inputs/Result Data_1
//     PlcTask Inputs/BarCodeReaders.BCR_S2150_01.ResultData @bit 80 <-> Connection 2 (Input/Output)/Inputs/Result Data_10
//     PlcTask Inputs/BarCodeReaders.BCR_S2150_01.ResultData @bit 88 <-> Connection 2 (Input/Output)/Inputs/Result Data_11
//     PlcTask Inputs/BarCodeReaders.BCR_S2150_01.ResultData @bit 96 <-> Connection 2 (Input/Output)/Inputs/Result Data_12
//     PlcTask Inputs/BarCodeReaders.BCR_S2150_01.ResultData @bit 104 <-> Connection 2 (Input/Output)/Inputs/Result Data_13
//     PlcTask Inputs/BarCodeReaders.BCR_S2150_01.ResultData @bit 112 <-> Connection 2 (Input/Output)/Inputs/Result Data_14
//     PlcTask Inputs/BarCodeReaders.BCR_S2150_01.ResultData @bit 120 <-> Connection 2 (Input/Output)/Inputs/Result Data_15
//     PlcTask Inputs/BarCodeReaders.BCR_S2150_01.ResultData @bit 128 <-> Connection 2 (Input/Output)/Inputs/Result Data_16
//     PlcTask Inputs/BarCodeReaders.BCR_S2150_01.ResultData @bit 136 <-> Connection 2 (Input/Output)/Inputs/Result Data_17
//     PlcTask Inputs/BarCodeReaders.BCR_S2150_01.ResultData @bit 144 <-> Connection 2 (Input/Output)/Inputs/Result Data_18
//     PlcTask Inputs/BarCodeReaders.BCR_S2150_01.ResultData @bit 152 <-> Connection 2 (Input/Output)/Inputs/Result Data_19
//     PlcTask Inputs/BarCodeReaders.BCR_S2150_01.ResultData @bit 16 <-> Connection 2 (Input/Output)/Inputs/Result Data_2
//     PlcTask Inputs/BarCodeReaders.BCR_S2150_01.ResultData @bit 160 <-> Connection 2 (Input/Output)/Inputs/Result Data_20
//     PlcTask Inputs/BarCodeReaders.BCR_S2150_01.ResultData @bit 168 <-> Connection 2 (Input/Output)/Inputs/Result Data_21
//     PlcTask Inputs/BarCodeReaders.BCR_S2150_01.ResultData @bit 176 <-> Connection 2 (Input/Output)/Inputs/Result Data_22
//     PlcTask Inputs/BarCodeReaders.BCR_S2150_01.ResultData @bit 184 <-> Connection 2 (Input/Output)/Inputs/Result Data_23
//     PlcTask Inputs/BarCodeReaders.BCR_S2150_01.ResultData @bit 192 <-> Connection 2 (Input/Output)/Inputs/Result Data_24
//     PlcTask Inputs/BarCodeReaders.BCR_S2150_01.ResultData @bit 200 <-> Connection 2 (Input/Output)/Inputs/Result Data_25
//     PlcTask Inputs/BarCodeReaders.BCR_S2150_01.ResultData @bit 24 <-> Connection 2 (Input/Output)/Inputs/Result Data_3
//     PlcTask Inputs/BarCodeReaders.BCR_S2150_01.ResultData @bit 32 <-> Connection 2 (Input/Output)/Inputs/Result Data_4
//     PlcTask Inputs/BarCodeReaders.BCR_S2150_01.ResultData @bit 40 <-> Connection 2 (Input/Output)/Inputs/Result Data_5
//     PlcTask Inputs/BarCodeReaders.BCR_S2150_01.ResultData @bit 48 <-> Connection 2 (Input/Output)/Inputs/Result Data_6
//     PlcTask Inputs/BarCodeReaders.BCR_S2150_01.ResultData @bit 56 <-> Connection 2 (Input/Output)/Inputs/Result Data_7
//     PlcTask Inputs/BarCodeReaders.BCR_S2150_01.ResultData @bit 64 <-> Connection 2 (Input/Output)/Inputs/Result Data_8
//     PlcTask Inputs/BarCodeReaders.BCR_S2150_01.ResultData @bit 72 <-> Connection 2 (Input/Output)/Inputs/Result Data_9
//     PlcTask Inputs/BarCodeReaders.BCR_S2150_01.ResultID <-> Connection 2 (Input/Output)/Inputs/Result ID
//     PlcTask Inputs/BarCodeReaders.BCR_S2150_01.ResultLength <-> Connection 2 (Input/Output)/Inputs/Result Length
//     PlcTask Inputs/BarCodeReaders.BCR_S2150_01.ResultsAvail <-> Connection 2 (Input/Output)/Inputs/Results Available
//     PlcTask Inputs/BarCodeReaders.BCR_S2150_01.TriggerAck <-> Connection 2 (Input/Output)/Inputs/Trigger Ack
//     PlcTask Inputs/BarCodeReaders.BCR_S2150_01.TriggerID <-> Connection 2 (Input/Output)/Inputs/Trigger ID
//     PlcTask Inputs/BarCodeReaders.BCR_S2150_01.TriggerReady <-> Connection 2 (Input/Output)/Inputs/Trigger Ready
//     PlcTask Outputs/BarCodeReaders.BCR_S2150_01.ResultsAck <-> Connection 2 (Input/Output)/Outputs/Results Ack
//     PlcTask Outputs/BarCodeReaders.BCR_S2150_01.Trigger <-> Connection 2 (Input/Output)/Outputs/Trigger
//     PlcTask Outputs/BarCodeReaders.BCR_S2150_01.TriggerEnable <-> Connection 2 (Input/Output)/Outputs/Trigger Enable
//   Building_1_5_Totes_ARUP Instance <-> Device 4 (TC3 EIP Scanner)/BCR_S3080_01
//     PlcTask Inputs/BarCodeReaders.BCR_S3080_01.Acquiring <-> Connection 2 (Input/Output)/Inputs/Acquiring
//     PlcTask Inputs/BarCodeReaders.BCR_S3080_01.DecodeComplete <-> Connection 2 (Input/Output)/Inputs/Decode Complete
//     PlcTask Inputs/BarCodeReaders.BCR_S3080_01.Decoding <-> Connection 2 (Input/Output)/Inputs/Decoding
//     PlcTask Inputs/BarCodeReaders.BCR_S3080_01.DeviceState <-> Inputs/State
//     PlcTask Inputs/BarCodeReaders.BCR_S3080_01.ResultCode <-> Connection 2 (Input/Output)/Inputs/Result Code
//     PlcTask Inputs/BarCodeReaders.BCR_S3080_01.ResultData <-> Connection 2 (Input/Output)/Inputs/Result Data
//     PlcTask Inputs/BarCodeReaders.BCR_S3080_01.ResultData @bit 8 <-> Connection 2 (Input/Output)/Inputs/Result Data_1
//     PlcTask Inputs/BarCodeReaders.BCR_S3080_01.ResultData @bit 80 <-> Connection 2 (Input/Output)/Inputs/Result Data_10
//     PlcTask Inputs/BarCodeReaders.BCR_S3080_01.ResultData @bit 88 <-> Connection 2 (Input/Output)/Inputs/Result Data_11
//     PlcTask Inputs/BarCodeReaders.BCR_S3080_01.ResultData @bit 96 <-> Connection 2 (Input/Output)/Inputs/Result Data_12
//     PlcTask Inputs/BarCodeReaders.BCR_S3080_01.ResultData @bit 104 <-> Connection 2 (Input/Output)/Inputs/Result Data_13
//     PlcTask Inputs/BarCodeReaders.BCR_S3080_01.ResultData @bit 112 <-> Connection 2 (Input/Output)/Inputs/Result Data_14
//     PlcTask Inputs/BarCodeReaders.BCR_S3080_01.ResultData @bit 120 <-> Connection 2 (Input/Output)/Inputs/Result Data_15
//     PlcTask Inputs/BarCodeReaders.BCR_S3080_01.ResultData @bit 128 <-> Connection 2 (Input/Output)/Inputs/Result Data_16
//     PlcTask Inputs/BarCodeReaders.BCR_S3080_01.ResultData @bit 136 <-> Connection 2 (Input/Output)/Inputs/Result Data_17
//     PlcTask Inputs/BarCodeReaders.BCR_S3080_01.ResultData @bit 144 <-> Connection 2 (Input/Output)/Inputs/Result Data_18
//     PlcTask Inputs/BarCodeReaders.BCR_S3080_01.ResultData @bit 152 <-> Connection 2 (Input/Output)/Inputs/Result Data_19
//     PlcTask Inputs/BarCodeReaders.BCR_S3080_01.ResultData @bit 16 <-> Connection 2 (Input/Output)/Inputs/Result Data_2
//     PlcTask Inputs/BarCodeReaders.BCR_S3080_01.ResultData @bit 160 <-> Connection 2 (Input/Output)/Inputs/Result Data_20
//     PlcTask Inputs/BarCodeReaders.BCR_S3080_01.ResultData @bit 168 <-> Connection 2 (Input/Output)/Inputs/Result Data_21
//     PlcTask Inputs/BarCodeReaders.BCR_S3080_01.ResultData @bit 176 <-> Connection 2 (Input/Output)/Inputs/Result Data_22
//     PlcTask Inputs/BarCodeReaders.BCR_S3080_01.ResultData @bit 184 <-> Connection 2 (Input/Output)/Inputs/Result Data_23
//     PlcTask Inputs/BarCodeReaders.BCR_S3080_01.ResultData @bit 192 <-> Connection 2 (Input/Output)/Inputs/Result Data_24
//     PlcTask Inputs/BarCodeReaders.BCR_S3080_01.ResultData @bit 200 <-> Connection 2 (Input/Output)/Inputs/Result Data_25
//     PlcTask Inputs/BarCodeReaders.BCR_S3080_01.ResultData @bit 24 <-> Connection 2 (Input/Output)/Inputs/Result Data_3
//     PlcTask Inputs/BarCodeReaders.BCR_S3080_01.ResultData @bit 32 <-> Connection 2 (Input/Output)/Inputs/Result Data_4
//     PlcTask Inputs/BarCodeReaders.BCR_S3080_01.ResultData @bit 40 <-> Connection 2 (Input/Output)/Inputs/Result Data_5
//     PlcTask Inputs/BarCodeReaders.BCR_S3080_01.ResultData @bit 48 <-> Connection 2 (Input/Output)/Inputs/Result Data_6
//     PlcTask Inputs/BarCodeReaders.BCR_S3080_01.ResultData @bit 56 <-> Connection 2 (Input/Output)/Inputs/Result Data_7
//     PlcTask Inputs/BarCodeReaders.BCR_S3080_01.ResultData @bit 64 <-> Connection 2 (Input/Output)/Inputs/Result Data_8
//     PlcTask Inputs/BarCodeReaders.BCR_S3080_01.ResultData @bit 72 <-> Connection 2 (Input/Output)/Inputs/Result Data_9
//     PlcTask Inputs/BarCodeReaders.BCR_S3080_01.ResultID <-> Connection 2 (Input/Output)/Inputs/Result ID
//     PlcTask Inputs/BarCodeReaders.BCR_S3080_01.ResultLength <-> Connection 2 (Input/Output)/Inputs/Result Length
//     PlcTask Inputs/BarCodeReaders.BCR_S3080_01.ResultsAvail <-> Connection 2 (Input/Output)/Inputs/Results Available
//     PlcTask Inputs/BarCodeReaders.BCR_S3080_01.TriggerAck <-> Connection 2 (Input/Output)/Inputs/Trigger Ack
//     PlcTask Inputs/BarCodeReaders.BCR_S3080_01.TriggerID <-> Connection 2 (Input/Output)/Inputs/Trigger ID
//     PlcTask Inputs/BarCodeReaders.BCR_S3080_01.TriggerReady <-> Connection 2 (Input/Output)/Inputs/Trigger Ready
//     PlcTask Outputs/BarCodeReaders.BCR_S3080_01.ResultsAck <-> Connection 2 (Input/Output)/Outputs/Results Ack
//     PlcTask Outputs/BarCodeReaders.BCR_S3080_01.Trigger <-> Connection 2 (Input/Output)/Outputs/Trigger
//     PlcTask Outputs/BarCodeReaders.BCR_S3080_01.TriggerEnable <-> Connection 2 (Input/Output)/Outputs/Trigger Enable

CONFIGURATION Building_1_5_Totes_ARUP
    RESOURCE PLC ON TwinCAT3
        TASK PlcTask(INTERVAL := T#10ms, PRIORITY := 20);
        PROGRAM MAIN WITH PlcTask : MAIN;
    END_RESOURCE
END_CONFIGURATION

// ---- DUTs/EAP/E_EAP_PubType.TcDUT
{attribute 'qualified_only'}
{attribute 'strict'}
TYPE E_EAP_PubType :
(
	e_AmsNetID 	:= 0,
	e_IPAddr	:= 1,
	e_MAC_ID	:= 2
);
END_TYPE

// ---- DUTs/EAP/ST_EAP_DEVICE.TcDUT
{attribute 'OPC.UA.DA' := '1'}
TYPE ST_EAP_DEVICE :
STRUCT
	DevName				:	STRING;		// Name of the EAP Device
	NetID				: 	STRING;		// Net ID of the EAP Device
	DevState	AT %I*	: 	UINT;		// EAP Device State
	DevCtrl		AT %Q*	: 	UINT;		// EAP Device Control
	Publisher			: 	ST_EAP_Publisher;		// Assumes single EAP to Publisher relationship
	Subscriber			: 	ST_EAP_Subscriber;		// Assumes single EAP to Subscriber relationship
END_STRUCT
END_TYPE

// ---- DUTs/EAP/ST_EAP_Publisher.TcDUT
TYPE ST_EAP_Publisher :
STRUCT
	Name				: 	STRING;		// Name of the EAP Publisher
	FrameState	AT %I*	: 	UINT;		// EAP FrameState, FrameState.0 = Not Transmitting, .1 = Frame too large, .2 = Subscriber Miissing
	FrameCtrl	AT %Q*	: 	UINT;		// EAP FrameCtrl, FrameCtrl.0 = Disable Sending, .1 = Remove destination MAC from ARP
	PubType				:	E_EAP_PubType := 0;	// EAP Publisher Type, AMS NetID (0), IP Address (1), MAC ID (2)
	NetID		AT %Q*	: 	AMSNETID;	// EAP Changeable NetID
	IPAddr		AT %Q*	: 	UDINT;		// EAP Changeable IP, stored as a single UDINT
	HMI_IPAddr			: 	USINTARR4;	// Used to enter IP Address on the HMI, MEMCPY function copies array to IPAddr 
	HMI_IPAddrDisp		: 	USINTARR4;	// Used to Display IP Address on the HMI, MEMCPY function copies IPAddr to Array 
	MACID		AT %Q*	: 	USINTARR6;	// EAP Changeable MAC ID, stored as an array of 6 USINT
	Variables			:	ARRAY[0..9] OF ST_EAP_Pub_Variable;		// Array of Published variables
END_STRUCT
END_TYPE

// ---- DUTs/EAP/ST_EAP_Pub_Variable.TcDUT
TYPE ST_EAP_Pub_Variable :
STRUCT
	Name				: 	STRING;		// Name of the Variable
	VarState	AT %I*	:	UINT;		// VarState.0 = Not Sent, 1 = Transmission Suspended, 0 = Transmission OK
	VarID 		AT %Q*	:	UINT;		// Changeable ID of the variable
	VarCtrl		AT %Q*	:	UINT;		// VarCtrl.0 = Disable publishing
END_STRUCT
END_TYPE

// ---- DUTs/EAP/ST_EAP_Subscriber.TcDUT
TYPE ST_EAP_Subscriber :
STRUCT
	Name				: 	STRING;		// Name of the EAP Subscriber
	FrameState	AT %I*	:	UINT;		// EAP FrameState, unused
	FrameCtrl	AT %Q*	:	UINT;		// EAP FrameCtrl, unused
	Variables			:	ARRAY[0..9] OF ST_EAP_Sub_Variable;		// Array of Subscribed variables
END_STRUCT
END_TYPE

// ---- DUTs/EAP/ST_EAP_Sub_Variable.TcDUT
TYPE ST_EAP_Sub_Variable :
STRUCT
	Name				: 	STRING;		// Name of the Variable
	VarState	AT %I*	:	UINT;		// VarState.0 = Invalid Hash/Version, .1 = Invalid Variable Length
	Quality		AT %I*	:	UINT;		// <>0, Duration the variable is not refreshed (in 100µs)
	CycleIndex	AT %I*	:	UINT;		// Incremented each publisher cycle
	VarId		AT %Q*	:	UINT;		// Changable Variable ID
	VarCtrl		AT %Q*	:	UINT;		// VarCtrl.1 = Ignore Hash/Version
END_STRUCT
END_TYPE

// ---- DUTs/E_EquipType.TcTLEO
{attribute 'qualified_only'}
{attribute 'strict'}
TYPE E_EquipType :
(
	Unknown := 0,
	System := 1,
	Conveyor := 2,
	Merge := 3,
	Gripper_SA := 4,
	Gripper_DA :=5,
	PinStop := 6,
	Pusher := 7,
	Divert := 8
) DINT;
END_TYPE

// ---- DUTs/E_StatusCode.TcDUT
{attribute 'qualified_only'}
{attribute 'strict'}
(*
	0-19 	-System level faults
	20-39	-Sorter Transfer Specific Status Codes
	40-59	-Diverter Transfer Specific Status Codes
	60-79	-Transfer Specific Status Codes
*)
TYPE E_StatusCode :
(
	No_Status				:= 0,
	OK						:= 1,
	Stopped					:= 2,
	Faulted					:= 3,	
	UnknownError	 		:= 9,	
	
	NotInSorter				:= 20,	
	UpdateRequested			:= 21,
	QueryNeeded				:= 22,
	UpdateNeeded 			:= 23,
	UpdateReceived 			:= 24,
	ReqNotReceived			:= 25,
	ItemNotUpdated			:= 26,
	UnidentifiedItem		:= 27,
	ItemNotFound			:= 28,
	Sorter_UnknownError 	:= 29,
	Assign_Accepted			:= 30,
	Assign_Full				:= 31,
	Assign_NotFound			:= 32,
	Assign_NotInducted		:= 33,
	Exiting_Sorter			:= 34,
	Exited_Sorter			:= 35,
	
	Divert_Idle				:= 40,
	In_Sorter 				:= 41,
	Diverting 				:= 42,
	Divert_Missed 			:= 43,
	Divert_Full				:= 44,
	Divert_Offline			:= 45,
	Divert_Faulted			:= 46,
	Divert_NotInducted		:= 47,
	Divert_LateAssignment	:= 48,
	Divert_UnknownError 	:= 49,
	Divert_Recirculated		:= 50,
	Divert_Detected			:= 51,
	Divert_Success			:= 52,
	Divert_Complete			:= 53,
	
	In_Transfer 			:= 61,
	Transferring 			:= 62,
	Tranfer_Success	 		:= 63,
	Transfer_Missed 		:= 64,
	Transfer_Failed 		:= 65,	
	Transfer_UnknownError 	:= 69
) USINT;
END_TYPE

// ---- DUTs/Messages/E_EquipmentUpdate.TcTLEO
{attribute 'qualified_only'}
{attribute 'strict'}
TYPE E_EquipmentUpdate :
(
	Manual := 1,
	Auto := 2,
	Offline := 3,
	Running := 4,
	SleepActive := 5,
	Faulted := 6,
	OverHeight := 7
);
END_TYPE

// ---- DUTs/Messages/E_MessageIds.TcTLEO
//{attribute 'qualified_only'}
{attribute 'strict'}
TYPE E_MessageIds :
(
	NoMessage_00 := 0,
	TransportCommand_05 := 5,
	LocationUpdateResponse_07 := 7,
	EquipmentStatusResponse_08 := 8,
	KeepAlive_09 := 9,
	Arrival_23 := 23,
	TransportResponse_25 := 25,
	TransportComplete_26 := 26,
	LocationUpdate_27 := 27,
	EquipmentStatusUpdate_28 := 28,
	KeepAliveResponse_29 := 29
);
END_TYPE

// ---- DUTs/Messages/E_TransportComplete.TcDUT
{attribute 'qualified_only'}
{attribute 'strict'}
TYPE E_TransportComplete :
(
	Success := 0,
	Unavailable := 1,
	Faulted := 2,
	Offline := 3,
	Passed := 8,
	ConfirmFailed := 11,
	InductFailed := 12
)INT ;
END_TYPE

// ---- DUTs/Messages/E_TransportResponse.TcTLEO
{attribute 'qualified_only'}
{attribute 'strict'}
TYPE E_TransportResponse :
(
	Accepted := 0,
	DivertLaneUnavailable := 1,
	LoadIdNotFound := 2,
	UnknownFailure := 11,
	NextLoadReady := 12,
	LateInduction := 13
);
END_TYPE

// ---- DUTs/Messages/ST_Msg_ConveyorStat.TcDUT
TYPE ST_Msg_ConveyorStat :
STRUCT
	DeviceID:	STRING(5);
	Status:	INT;
END_STRUCT
END_TYPE

// ---- DUTs/Messages/ST_Msg_EquipStat.TcDUT
TYPE ST_Msg_EquipStat :
STRUCT
	DeviceID:	STRING(5);
	Status:	INT;
END_STRUCT
END_TYPE

// ---- DUTs/ST_EquipmentStatus.TcDUT
TYPE ST_EquipmentStatus :
STRUCT
	Sts_EquipmentState:	ST_StateCntrlSts;		// State Status
	Sts_SleepingActive: BOOL;	// Status to show conveyor is in sleep state
	Sts_All_Intlks_OK:	BOOL;		// Status bit to show that all interloks are good to Run 
	Sts_FaultActive:	BOOL;	// Status Bit Showing that a fault is present (0= No Active Faults, 1= Fault Active)
	Sts_WarnActive:	BOOL;	// Status Bit Showing that a warning is present (0= No Active Warnings, 1= Warning Active)
	Sts_All_Evnts_OK: BOOL;		// Status Bit Showing that ALL Events are OK to RUN (0= Event Present, 1= OK to Run)
	Sts_IsRunning :BOOL;	// Status to show conveyor is running (1=running)
	Sts_IsExtending :BOOL;	// Status to show Actuator is extending (1=extending)
	Sts_IsExtended :BOOL;	// Status to show Actuator is extended (1=extended)
	Sts_IsRetracting :BOOL;	// Status to show Actuator is retracting (1=retracting)
	Sts_IsRetracted :BOOL;	// Status to show Actuator is retracted (1=retracted)
END_STRUCT
END_TYPE

// ---- DUTs/ST_SafetyState.TcDUT
TYPE ST_SafetyState :
STRUCT
	Reset 	 	AT %Q* : BOOL;
	Run 	 	AT %Q* : BOOL;
	ErrAck 	 	AT %Q* : BOOL;
	CommErrAck	AT %Q*	:BOOL;
	ComErr    	AT %I* : BOOL;
	FBErr     	AT %I* : BOOL;
	OtherErr  	AT %I* : BOOL;
	InRun 		AT %I* : BOOL;
END_STRUCT
END_TYPE

// ---- FunctionBlocks/Binder/DUTs/ST_Binder.TcDUT
{attribute 'OPC.UA.DA' := '1'}
TYPE ST_Binder :
STRUCT
	State		:	ST_BinderState;		// State of the Binder
	FromBinder	:	ST_FromBinder;		// Data Recevied from the Binder
	ToBinder	:	ST_ToBinder;		// Data Sent to the Binder
END_STRUCT
END_TYPE

// ---- FunctionBlocks/Binder/DUTs/ST_BinderState.TcDUT
TYPE ST_BinderState :
STRUCT
	DoorOpenOK  	AT %I*: BOOL;
	EstopOK  		AT %I*: BOOL;
	NetReset		AT %I*: BOOL;
	VlvBankPower 	AT %I*: BOOL;
	DumpValve 		AT %I*: BOOL;
	SystemEstopOK	AT %I*: BOOL;
END_STRUCT
END_TYPE

// ---- FunctionBlocks/Binder/DUTs/ST_FromBinder.TcDUT
TYPE ST_FromBinder :
STRUCT
	ProcessingComplete :BOOL;
	Online: BOOL;
	RackProcessing : BOOL;
END_STRUCT
END_TYPE

// ---- FunctionBlocks/Binder/DUTs/ST_ToBinder.TcDUT
TYPE ST_ToBinder :
STRUCT
	ProductHeld : BOOL;
	StatusSingulator : UINT;
END_STRUCT
END_TYPE

// ---- FunctionBlocks/Conveyance/DUTs/E_ConvType.TcDUT
{attribute 'qualified_only'}
{attribute 'strict'}
TYPE E_ConvType :
(
	standard 	:= 0,
	end			:= 1,
	slave		:= 2
);
END_TYPE

// ---- FunctionBlocks/Divert/DUTs/ST_Divert.TcDUT
{attribute 'OPC.UA.DA' := '1'}
TYPE ST_Divert :
STRUCT
	{attribute 'OPC.UA.DA' := '0'}
	Config			: ST_DivertCfg;		// Configuration Variables

	Full 			: BOOL;				//Diverter full photo eye is blocked
	Jammed 			: BOOL;				//Jammed photo eye is blocked
	Faulted 		: BOOL;				//Returned faulted status
	Available 		: BOOL;				//Return availability status, auto/running/etc.  Will depend on the system and requirements

	Status 			: E_StatusCode := E_StatusCode.Divert_Idle; 	//Status Code, initialized to Idle

	ConfirmPE	   	: BOOL;				//Physical input address of photo eye
	FullPE		   	: BOOL;				//Physical input address of photo eye
	JamPE		   	: BOOL;				//Physical input address of photo eye 
	Output1	 		: BOOL;				//Physical output address of diverter
	Output2	  		: BOOL;				//Physical output address of diverter
	
	{attribute 'OPC.UA.DA' := '0'}
	Output1Flag		: DINT;				//Indicates what the encoder count is when output is energized
	
	FullTime		: TIME;				//Time that full PE has to be high before the lane is considered full     
	{attribute 'OPC.UA.DA' := '0'}
	FullTimer		: TON; 				//Timer that is used for checking how long the full PE is on
	
	{attribute 'OPC.UA.DA' := '0'}
	Item			: ST_Item;			// Currently Diverting Item
END_STRUCT
END_TYPE

// ---- FunctionBlocks/Divert/DUTs/ST_DivertCfg.TcDUT
{attribute 'OPC.UA.DA' := '1'}
TYPE ST_DivertCfg :
STRUCT
	ID 				: STRING;			// User assigned Divert indetifier		
	EquipID 		: STRING[5];		// Identifier used for host communication		
	Number			: INT;				// Divert number, can be distinct from the Index in the Divert Array
	Distance		: INT;				// Distance, in encoder counts, from induct photo eye
	ConfirmDist		: INT;				// Distance from the Divert point to the Confirm PE
	Direction		: BOOL;				// 0 = Divert to one side, 1 = Divert to the other side 
	FullTime		: REAL;				// Time, in seconds, that full PE has to be high before the lane is considered full
	IsDischarge		: BOOL;				// TRUE, process and test for items destined for non-discharge diverts that missed
END_STRUCT
END_TYPE

// ---- FunctionBlocks/Encoder/DUTs/ST_Encoder.TcDUT
TYPE ST_Encoder :
STRUCT
	EncoderRawCount : UDINT;	// Raw encoder Count, acommodates 16 and 32 bit encoder resoultions
	CurrentCount : UDINT;		// Current Pulse Count
	BitMaskSize	: UINT;			// Number of bits to mask into the CurrentCount from the Actual Encoder Pulses
	EncoderString	: STRING;	// Encoder pulses formatted as string
END_STRUCT
END_TYPE

// ---- FunctionBlocks/FB_Merge/E_MergeState.TcDUT
{attribute 'qualified_only'}
//{attribute 'strict'}
TYPE E_MergeState :
(
	stStopped := 0,
	stClearTakeAway := 1,
	stMergeOperational := 2,
	stMergeManual := 3
)INT;
END_TYPE

// ---- FunctionBlocks/FB_Merge/Merge Inlet/ST_MergeInlet.TcDUT
{attribute 'OPC.UA.DA' := '1'}
TYPE ST_MergeInlet :
STRUCT
	{attribute 'OPC.UA.DA' := '0'}
	Cfg		:	ST_MergeInletCfg;
	Ctrl	:	ST_MergeInletCtrl;
END_STRUCT
END_TYPE

// ---- FunctionBlocks/FB_Merge/Merge Inlet/ST_MergeInletCfg.TcDUT
{attribute 'OPC.UA.DA' := '1'}
TYPE ST_MergeInletCfg :
STRUCT
	Cfg_UseMtrFdBck				:	BOOL := FALSE;	// Configuration bit to determine if motor feed back is used (1= use feedback)
	Cfg_UseHighWaterPE			:	BOOL := FALSE;	// Configuration bit to determine if the High Water indicator PE is used (1= use High Water PE)
	Cfg_UseHiHiWaterPE			:	BOOL := FALSE;	// Configuration bit to determine if the HiHi Water indicator PE is used (1= use HiHi Water PE)
	Cfg_HighTriggerTime			:	REAL := 1;		// Time that full trigger has to be on to record high condition
	Cfg_HiHiTriggerTime			:	REAL := 1;		// Time that full trigger has to be on to record hihi condition
	Cfg_HiHiClearTime			:	REAL := 10;		// Time Merge runs in response to a HiHi Water condition
	Cfg_MrgReqPrdctWaitTime		: 	REAL := 45;		// Time that product has to wait for full mark to be reached before requesting merge
	Cfg_ReleaseCount			:	INT := 1;		// Required count to be released before switching merge locations
	Cfg_ReleaseCountWaitTime	:	REAL := 60;		// Time to wait to achieve release count before switching merge locations
	Cfg_ClearRunOutTime			:	REAL := 25;		// Time to wait for product to clear the merge
	Cfg_MergeName				:	STRING(20);		// Name used to Identify the Merge on the HMI
END_STRUCT
END_TYPE

// ---- FunctionBlocks/FB_Merge/Merge Inlet/ST_MergeInletCtrl.TcDUT
{attribute 'OPC.UA.DA' := '1'}
TYPE ST_MergeInletCtrl :
STRUCT
	PhotoEyeDischarge			:	BOOL;			// Photo Eye at the discharge of the assigned merge location
	PhotoEyeEntryHigh			:	BOOL;			// Photo Eye at the Full (high water) location of the merge
	PhotoEyeEntryHiHi			:	BOOL;			// Photo Eye at the Full (hihi water) location of the merge
	MergeInletMtrFdBck			:	BOOL;			// Current motor feedback for the assigned merge location
	In_InletState				:	E_StateCntrl;	// The State of the merge take away conveyor
	In_oMergeRelease			:	BOOL;
	{attribute 'OPC.UA.DA' := '0'}
	SimActive					:	BOOL;			// Simulation Bit 
END_STRUCT
END_TYPE

// ---- FunctionBlocks/FB_Merge/Merge Inlet/ST_MergeInletSts.TcDUT
{attribute 'OPC.UA.DA' := '1'}
TYPE ST_MergeInletSts :
STRUCT
	MergeRequested				:	BOOL;		// Merge has been Requested (1=request Active)
	Granted						:	BOOL;		// The Granted state of this Inlet
	MergeComplete				:	BOOL;		// Flag to finish merging
	HiHiDetected				:	BOOL;		// HiHi Event has been detected and requires control
	HiHiTimedReleaseActive		:	BOOL;		// Indicates that a HiHi event clearout is in process
	Out_MergeInletRunActive		:	BOOL;		// Output for Merge inlet run
	Sts_MergeInletRun			:	BOOL;		// Merge Inlet status Motor is currently running (1=merging or running)
	MergeRunOutActive			:	BOOL;		// Flag to indicate that the Merge Run Out is active (1=active)
	CrrntReleaseCount			:	INT;		// The current count of product released
END_STRUCT
END_TYPE

// ---- FunctionBlocks/FB_Merge/ST_MergeSts.TcDUT
{attribute 'OPC.UA.DA' := '1'}
TYPE ST_MergeSts :
STRUCT
	MergeEnabled			: 	BOOL;		// Merge is enabled 
	MergeTakeAwayMtrActive	:	BOOL;		// Output for Merge take away motor
	MergeSubState			:	E_MergeState;
	MergeSubStateTxt		:	STRING(20);
	MergeJammed				:	BOOL;		// Merge is Jammed
	InletCount				:	INT;
END_STRUCT
END_TYPE

// ---- FunctionBlocks/FB_MotionMerge/ST_MotionMergeConfig.TcDUT
{attribute 'OPC.UA.DA' := '1'}
TYPE ST_MotionMergeConfig :
STRUCT
	MergeDistance: 			UINT;	// The distance from the induct PE to the merge point (Merge start location)
	MergeClearDistance: 	UINT;	// The distance from the induct PE to a cleared point past the merge (Merge end location)
	MergeOpening_Min: 		UINT;	// The minimum window size to allow a merge
	Item_ExtendFwd:			UINT;	// The distance to Extend the Item lead edge
	Item_ExtendRev:			UINT;	// The distance to Extend teh Item Trail edge
	MergeClearTime: 		REAL;	// The time, in seconds, to declare the merge clear
END_STRUCT
END_TYPE

// ---- FunctionBlocks/FB_MotionMerge/ST_MotionMergeItem.TcDUT
TYPE ST_MotionMergeItem :
STRUCT
	Count_InductStart	: UDINT;
	Count_InductEnd	: UDINT;
	Length	: UDINT;
	OnConveyor	: BOOL;
END_STRUCT
END_TYPE

// ---- FunctionBlocks/Item/DUTs/ST_Item.TcDUT
TYPE ST_Item :
STRUCT
	ID : STRING := '';		// Bar Code 	
	UniqueID : DINT := 0;		// Generic ID for tracking
	Destination : DINT := 0;
	DestinationIdx : DINT := 0;
	Length : DINT := 0;
	Status : E_StatusCode := E_StatusCode.No_Status;
	ExtStatus : E_StatusCode := E_StatusCode.No_Status;
	CapturedInMetrics : BOOL;
	DeviceID:	STRING(5);	// Device ID associated with this record
	MessageType:	E_MessageIds;	// Message Type associated with this record
END_STRUCT
END_TYPE

// ---- FunctionBlocks/Item/DUTs/ST_ItemBuffer.TcDUT
TYPE ST_ItemBuffer :
STRUCT
	aBufferData	: ARRAY [0..99] OF ST_Item;	// Data stored in the buffer, 100 elements
	nInPointer	: UDINT;						// Pointer for data put into the buffer
	bClear		: BOOL;							// Clear the Buffer
END_STRUCT
END_TYPE

// ---- FunctionBlocks/Item/DUTs/ST_ItemBufferFdbk.TcDUT
TYPE ST_ItemBufferFdbk :
STRUCT
	bEmpty		: BOOL;							// Buffer is Empty
END_STRUCT
END_TYPE

// ---- FunctionBlocks/Item/DUTs/ST_ItemLogBuffer.TcDUT
TYPE ST_ItemLogBuffer :
STRUCT
	aBufferData	:	ARRAY [0..999] OF ST_Item;	// Data stored in the buffer, 100 elements
	nInPointer	:	UDINT;							// Pointer for data put into the buffer
END_STRUCT
END_TYPE

// ---- FunctionBlocks/Item/DUTs/ST_ItemTemporary.TcDUT
TYPE ST_ItemTemporary :
STRUCT
	Item	: ST_Item;
	Counts	: UDINT;
END_STRUCT
END_TYPE

// ---- FunctionBlocks/LEDControl/ST_HMILEDMode.TcDUT
{attribute 'OPC.UA.DA' := '1'}
TYPE ST_HMILEDMode :
STRUCT
	PB_ControlCnvyrsTogether:	BOOL;		// Bit tocontrol all conveyors together (0 = individual control, 1 = All controlled together)
	PB_SaveLEDConfig:	BOOL;		// Bool to Save current test configuration values to the mode array at indexed item
	PB_LoadDefaultLEDConfig:	BOOL;		// Bool to Reload default mode value into configuration array at indexed item
	PB_TestLEDConfig:	BOOL;		// Bit to turn on LED for testing
	ST_LEDConfig: ST_LEDMode;		// Values from HMI to configure LED Hue Values
	LaneValueLEDConfig:	BYTE;	// Value for mode configuration array index
	ModeValueLEDConfig:	BYTE;	// Value for mode configuration array index
	FlashValueLEDConfig:	BYTE;	// Value for flash mode configuration array at indexed item
END_STRUCT
END_TYPE

// ---- FunctionBlocks/LEDControl/ST_LEDMode.TcDUT
TYPE ST_LEDMode :
STRUCT
	Value1:	ST_RGB := (Value_Red := 0, Value_Green := 0, Value_Blue := 0);		// The LED Values for Color 1
	Value2:	ST_RGB := (Value_Red := 0, Value_Green := 0, Value_Blue := 0);		// The LED Values for Color 2
	Flashing:	BYTE;		// Value (Byte) to make light flash or not (0=Steady On, 1= Blinking Slow, 2= Blinking Fast)
	LabelText:	STRING(50);	// Label Text for Configuration Mode	
END_STRUCT
END_TYPE

// ---- FunctionBlocks/LEDControl/ST_RGB.TcDUT
TYPE ST_RGB :
STRUCT
	Value_Red:	BYTE;		// The Value for the Red LED (0=Off, 255 = Full on)
	Value_Green:	BYTE;		// The Value for the Blue LED (0=Off, 255 = Full on)
	Value_Blue:	BYTE;		// The Value for the Blue LED (0=Off, 255 = Full on)
END_STRUCT
END_TYPE

// ---- FunctionBlocks/Logging/ST_LogMsg.TcDUT
TYPE ST_LogMsg :
STRUCT
	DateandTime : STRING(24);
	Status : E_StatusCode; 
	StatusDescription : WSTRING;
	ItemID : DINT;
END_STRUCT
END_TYPE

// ---- FunctionBlocks/Server/Data types/E_ConnectionSteps.TcDUT
TYPE E_ConnectionSteps :
(
	eCONNECTION_STATE_IDLE,
	eCONNECTION_STATE_CONNECT_START,
	eCONNECTION_STATE_CONNECT_WAIT,
	eCONNECTION_STATE_DATAEXCHANGE,
	eCONNECTION_STATE_CLOSE_START,
	eCONNECTION_STATE_CLOSE_WAIT,
	eCONNECTION_STATE_ERROR
);
END_TYPE

// ---- FunctionBlocks/Server/Data types/E_ServerSteps.TcDUT
TYPE E_ServerSteps :
(
	eSERVER_STATE_IDLE,
	eSERVER_STATE_LISTENER_OPEN_START,
	eSERVER_STATE_LISTENER_OPEN_WAIT,
	eSERVER_STATE_REMOTE_CLIENTS_COMM,
	eSERVER_STATE_REMOTE_CLIENTS_CLOSE,
	eSERVER_STATE_LISTENER_CLOSE_START,
	eSERVER_STATE_LISTENER_CLOSE_WAIT,
	eSERVER_STATE_ERROR
);
END_TYPE

// ---- FunctionBlocks/Sorter/DUTs/ST_RoundRobin.TcDUT
TYPE ST_RoundRobin :
STRUCT
	Last_Enabled	:	UINT;
	Sent			:	UINT;
	{attribute 'OPC.UA.DA' := '0'}
	Config			:	ST_RoundRobinCfg;
END_STRUCT
END_TYPE

// ---- FunctionBlocks/Sorter/DUTs/ST_RoundRobinCfg.TcDUT
{attribute 'OPC.UA.DA' := '1'}
TYPE ST_RoundRobinCfg :
STRUCT
	Destination		:	DINT;
	Destinations	:	ARRAY [0..15] OF ST_RoundRobinDest;
END_STRUCT
END_TYPE

// ---- FunctionBlocks/Sorter/DUTs/ST_RoundRobinDest.TcDUT
TYPE ST_RoundRobinDest :
STRUCT
	Enabled			:	BOOL;
	Available		:	BOOL;
	aDestination	:	DINT;
END_STRUCT
END_TYPE

// ---- FunctionBlocks/Sorter/DUTs/ST_Sorter.TcDUT
{attribute 'OPC.UA.DA' := '1'}
TYPE ST_Sorter :
STRUCT
	{attribute 'OPC.UA.DA' := '0'}
	Config				: ST_SorterConfig;
	InductPE			: BOOL;
	EncoderCounts		: UDINT;
	LastUniqueID		: UINT;
	DischargePE			: BOOL;
	RoundRobin			: ST_RoundRobin;
END_STRUCT
END_TYPE

// ---- FunctionBlocks/Sorter/DUTs/ST_SorterConfig.TcDUT
{attribute 'OPC.UA.DA' := '1'}
TYPE ST_SorterConfig :
STRUCT
	Name				: STRING[5];
	EquipID				: STRING[5];
	Length				: UINT;
	InductWindow		: UINT;
	MinimumLength		: UINT;
	TailEndLength 		: UINT;
	Output2Offset		: UINT;
	DefaultDestination 	: DINT;
	DefaultDestIdx		: DINT;
	RecircDestination 	: DINT;
	RecircDestIdx 		: DINT;
	RecircUsed			: BOOL;
	RetainOnRestart		: BOOL;
	DivertCount			: DINT;
END_STRUCT
END_TYPE

// ---- FunctionBlocks/StateControl/E_OperStateCntrl.TcTLEO
{attribute 'qualified_only'}
// {attribute 'strict'}
TYPE E_OperStateCntrl :
(
	stopped:= 0,
	running:= 1,
	sleeping:= 2,
	overheight:= 3,
	extended := 4,
	extending := 5,
	retracted := 6,
	retracting := 7,
	unknown :=8,
	offline :=9,
	auto := 10,
	manual := 11,
	faulted	:= 12
) INT;
END_TYPE

// ---- FunctionBlocks/StateControl/E_StateCntrl.TcTLEO
{attribute 'qualified_only'}
// {attribute 'strict'}
TYPE E_StateCntrl :
(
	// Allowed to transition to Manual
	stOffline:= 0,
	// Allowed to transition to Manual/Faulted 
	stAuto:= 1,
	// Allowed to transition to Offline/Faulted/Manual 
	stManual:= 2,
	// Allowed to transition to Offline/Manual 
	stFaulted:= 3
) INT;
END_TYPE

// ---- FunctionBlocks/StateControl/E_StopCodes.TcTLEO
{attribute 'qualified_only'}
{attribute 'strict'}
TYPE E_StopCodes :
(
	NoStop := 0,
	SystemStop := 1,
	MotorOL := 2,
	VFD_Fault := 3,
	ProductJam := 4,
	MotorRunTO := 5,
	VFDRunTO := 6,
	LowAir := 7,
	MergeJam := 8,
	SlackBeltFault := 9,
	EncoderFault := 10,
	TransferTO := 11,
	TransferLP := 12,
	ActuatorTO := 13,
	SprialTorque := 14,
	DisconnectState := 15,
	ReleaseFault := 16,
	PanelIOFLT := 17,
	FieldIOFLT := 18,
	UnderHeightFLT := 19,
	OverHeightFLT := 20,
	Taper :=21,
	DeviceNoInAuto := 22
) UINT;
END_TYPE

// ---- FunctionBlocks/StateControl/ST_StateCntrlPB.TcDUT
TYPE ST_StateCntrlPB :
STRUCT
	OfflinePB:		BOOL;	// State control, take related equipment offline		
	AutoPB:			BOOL;	// State control, put related equipment into Automatic operation mode
	ManPB:			BOOL;	// State control, put related equipment into Maunual operation mode
	StopPB: 		BOOL;	// State control, Stop equipment, in manual, execute stop command, in auto, move equipment to manual and stop equipment
	ResetPB:		BOOL;	// State control, Reset any faults/warnings associated with the equipment
	ManMotorRunPB:	BOOL;	// State control, manually run motor 
	ManExtendPB:	BOOL;	// State control, manually execute actuator extend
	ManRetractPB:	BOOL;	// State control, manually execute actuator retract
END_STRUCT
END_TYPE

// ---- FunctionBlocks/StateControl/ST_StateCntrlSts.TcDUT
TYPE ST_StateCntrlSts :
STRUCT
	{attribute 'OPC.UA.DA' := '1'}
	CrntState:			E_StateCntrl;
	{attribute 'OPC.UA.DA' := '1'}
	CrntStateTxt:		STRING(20);				// The current state in text string
	{attribute 'OPC.UA.DA' := '0'}
	CrntOperState: 		E_OperStateCntrl;		// The Current Operational state
	{attribute 'OPC.UA.DA' := '0'}
	CrntOperStateTxt:	STRING(20);				// The current Operational state in text string
	{attribute 'OPC.UA.DA' := '0'}
	EquipType: 			DINT;					// Stores Enumeration type E_EquipType
	{attribute 'OPC.UA.DA' := '0'}
	Index: 				DINT;					// Local index assigned to this equipment
	{attribute 'OPC.UA.DA' := '0'}
	Label: 				STRING(20); 			// String value assigned to this equipment for status updates
	{attribute 'OPC.UA.DA' := '0'}
	RemIndex: 			DINT;					// Remote index assigned to this equipment, for system status monitoring
	{attribute 'OPC.UA.DA' := '0'}
	LstState:			E_StateCntrl;
	{attribute 'OPC.UA.DA' := '0'}
	LstOperState:		E_OperStateCntrl;
	{attribute 'OPC.UA.DA' := '0'}
	stsStopRegister: 	ARRAY[0..1] OF UDINT;	// Stop Register
	{attribute 'OPC.UA.DA' := '0'}
	StateRunOK:			BOOL;
	{attribute 'OPC.UA.DA' := '0'}
	StateChanged:		BOOL;					// Single scan output to show that state has changed
	{attribute 'OPC.UA.DA' := '0'}
	StsOffline:			BOOL;					// Output that shows State is Offline
	{attribute 'OPC.UA.DA' := '0'}
	StsAuto:			BOOL;					// Output that shows State is in Auto
	{attribute 'OPC.UA.DA' := '0'}
	StsMan:				BOOL;					// Output that shows State is in Manual
	{attribute 'OPC.UA.DA' := '0'}
	StsFaulted:			BOOL;					// Output that shows State is Faulted
	{attribute 'OPC.UA.DA' := '0'}
	StsHasWarnings: 	BOOL;					// Output that shows the Equipment has Warnings (Alerts)
	{attribute 'OPC.UA.DA' := '0'}
	Received:			ST_StateCntrlPB;		// Single scan outputs for possible push button events
	{attribute 'OPC.UA.DA' := '0'}
	RcvdFault:			BOOL;					// Single scan output to show input was received
//	RcvdOffline:		BOOL;					// Single scan output to show input was received
//	RcvdAuto:			BOOL;					// Single scan output to show input was received
//	RcvdManual:			BOOL;					// Single scan output to show input was received
//	RcvdReset:			BOOL;					// Single scan output to show input was received
//	RcvdStartPB:		BOOL;					// Single scan output to show input was received
//	RcvdStopPB:			BOOL;					// Single scan output to show input was received
END_STRUCT
END_TYPE

// ---- FunctionBlocks/Utils/Events/ST_CfgEvents.TcDUT
{attribute 'OPC.UA.DA' := '1'}
TYPE ST_CfgEvents :
STRUCT
	Description:	STRING(40);		// The Text Description of the Interlock/Event assigned to the corresponding Input
	DeviceLabel:	STRING(15);		// The Text Description or Label of the Interlock/Event Device assigned to the corresponding Input
	StopCode:	UINT;				// Stop Code associated with this Event
	EventDelay:	TIME;				// Allow an event to be delayed before being activated
	OKState:	BOOL;		// The OK state of the Interlock/Event or the state that is required to be "Alright to Run" (0 or 1)
	LatchRequired:	BOOL;		// Configuration Bit to set that the Interlock/Event Requires Latching until HMI_Reset (0 = NOT Latching, 1 = Latching)
	ByPssAllwd:	BOOL;		// Configuration bit to set if the Interlock/Event is able to be bypased or not( 0= Bypass Allowed, 1 = Bypass Not Allowed	
	HMI_BypassPB:	BOOL;		//Input for Individual Bypass Bits for each Interlock/Event (0= Bypass Not Active, 1 = Bypass Active)
	FaultWarn:	BOOL;		// // Configuration Bit to set if Event causes a Fault or Warning (0=Warning, 1=Fault) 
END_STRUCT
END_TYPE

// ---- FunctionBlocks/Utils/Events/ST_EventSts.TcDUT
{attribute 'OPC.UA.DA' := '1'}
TYPE ST_EventSts :
STRUCT
	Description:	STRING(30);		// The Text Description of the Interlock/Event assigned to the corresponding Input
	DeviceLabel:	STRING(15);		// The Text Description or Label of the Interlock/Event Device assigned to the corresponding Input
	Status:	BOOL;		// Event status 
	StatusTxt: STRING(10);
END_STRUCT
END_TYPE

// ---- FunctionBlocks/VFD/DUTs/DRIVE_STATE.TcTLEO
{attribute 'qualified_only'}
{attribute 'strict'}
TYPE DRIVE_STATE :
(
	SWITCH_ON_INHIBITED := 64,
	SWITCH_ON_INHIBITED_BIT_5 := 96,
	NOT_READY_TO_SWITCH_ON := 0,
	NOT_READY_TO_SWITCH_ON_BIT_5 := 32,
	READY_TO_SWITCH_ON := 33,
	SWITCHED_ON		   := 35,
	QUICK_STOP_ACTIVE	:= 7,
	OPERATION_ENABLED := 39,
	TROUBLE			:= 8,
	TROUBLE_BIT_5	:= 40,
	FAULT_REACTION_ACTIVE := 15,
	FAULT_REACTION_ACTIVE_BIT_5 := 47
) UINT;
END_TYPE

// ---- GVLs/GVL_EquipArrays.TcGVL
{attribute 'qualified_only'}
VAR_GLOBAL
	nEquipIndex : DINT := 0;	// Index used to Assign the Equipment Index for System Status Reporting
	nEquip_Count AT %Q* : DINT; //Count of Equipment to Process in System PLC
	{attribute 'OPC.UA.DA' := '0'}
	aEquipStatusArray_Out AT %Q* : ARRAY[1..cEQUIP_COUNT_MAX] OF ST_StateCntrlSts; //Array of Equipment Status Outbound
	{attribute 'OPC.UA.DA' := '0'}
	aEquipStatusArray_In AT %I* : ARRAY[1..cEQUIP_COUNT_MAX] OF ST_StateCntrlSts; //Array of Equipment Status Inbound
	
	// System Equipment
	nSystemEquip_Count : DINT; //Count of Equipment to Process in System PLC
	{attribute 'OPC.UA.DA' := '0'}
	aSystemEquipStatusArray : ARRAY[1..cEQUIP_COUNT_MAX] OF ST_StateCntrlSts; //Array of Equipment Status Current
	{attribute 'OPC.UA.DA' := '0'}
	aSystemEquipStatusArray_Last : ARRAY[1..cEQUIP_COUNT_MAX] OF ST_StateCntrlSts; //Array of Equipment Status Last State
END_VAR

VAR_GLOBAL CONSTANT
	cEQUIP_COUNT_MAX : DINT := 50;	//Adjust when adding equipment to monitor
END_VAR

// ---- GVLs/GVL_IO.TcGVL
{attribute 'qualified_only'}
VAR_GLOBAL
	INIT						: BOOL := TRUE;		// Initialization Bit
	
// ------ Note:	All Photo Eyes are defined and linked in the Photo Eye Function Block in PhotoEyes.PRG
// ------ Note:	All Prox Switches are defined and linked in the ProxSensors.PRG

	{attribute 'OPC.UA.DA' := '1'}
	PB_SysStart AT %I* 		:BOOL;		//System Start Button
	{attribute 'OPC.UA.DA' := '1'}
	PB_SysStop	AT %I*		:BOOL;		//System Stop Button
	{attribute 'OPC.UA.DA' := '1'}
	PB_SysReset	AT %I* 		:BOOL; 		//System Reset Button
	{attribute 'OPC.UA.DA' := '1'}
	PB_RemoteReset_3211 AT %I*		: BOOL;	//P2150 Reset Button
	{attribute 'OPC.UA.DA' := '1'}
	PB_RemoteReset_8251 AT %I*		: BOOL;	//P2150 Reset Button
	{attribute 'OPC.UA.DA' := '1'}
	PB_RemoteReset_10221 AT %I*		: BOOL;	//P2140 Reset Button
	
	
	{attribute 'OPC.UA.DA' := '1'}
	SystemAirPressure AT %I*	:BOOL;

	
	{attribute 'OPC.UA.DA' := '1'}
	HornMainPanel				AT %Q* 	:BOOL;	//Panel Tower Horn
	{attribute 'OPC.UA.DA' := '1'}
	LT_MainPanelStack_Red		AT %Q*	:BOOL;	//Panel	Tower Red Light
	{attribute 'OPC.UA.DA' := '1'}
	LT_MainPanelStack_Yellow	AT %Q*	:BOOL;	//Panel	Tower Yellow Light
	{attribute 'OPC.UA.DA' := '1'}
	LT_MainPanelStack_Green		AT %Q*	:BOOL;	//Panel	Tower Green Light
	
	{attribute 'OPC.UA.DA' := '1'}
	LT_3131_Red	    AT %Q*	:BOOL;	//Panel	Tower Red Light
	{attribute 'OPC.UA.DA' := '1'}
	LT_3151_Yellow	AT %Q*	:BOOL;	//Panel	Tower Yellow Light
	{attribute 'OPC.UA.DA' := '1'}
	LT_3201_Green	AT %Q*	:BOOL;	//Panel	Tower Green Light
	
	{attribute 'OPC.UA.DA' := '1'}
	LT_8181_Red	    AT %Q*	:BOOL;	//Panel	Tower Red Light
	{attribute 'OPC.UA.DA' := '1'}
	LT_8191_Yellow	AT %Q*	:BOOL;	//Panel	Tower Yellow Light
	{attribute 'OPC.UA.DA' := '1'}
	LT_8231_Green	AT %Q*	:BOOL;	//Panel	Tower Green Light
	
	{attribute 'OPC.UA.DA' := '1'}
	LT_10161_Red	    AT %Q*	:BOOL;	//Panel	Tower Red Light
	{attribute 'OPC.UA.DA' := '1'}
	LT_10171_Yellow	AT %Q*	:BOOL;	//Panel	Tower Yellow Light
	{attribute 'OPC.UA.DA' := '1'}
	LT_10201_Green	AT %Q*	:BOOL;	//Panel	Tower Green Light
	
		{attribute 'OPC.UA.DA' := '1'}
	PanelEstop_OK AT %I* : BOOL;
	{attribute 'OPC.UA.DA' := '1'}
	Remote_PullCord2150_OK AT %I*: BOOL;
	{attribute 'OPC.UA.DA' := '1'}
	Remote_PullCord2142_OK AT %I*: BOOL;
	
	
//---------------------------------Motor Outputs-------------------------------------------------
	{attribute 'OPC.UA.DA' := '1'}
	P2130_RUN            AT %Q*   :BOOL;    //P2130 Run Command
	{attribute 'OPC.UA.DA' := '1'}
	P2135_RUN            AT %Q*   :BOOL;    //P2135 Run Command
	{attribute 'OPC.UA.DA' := '1'}
	P2140_RUN            AT %Q*   :BOOL;    //P2140 Run Command
	{attribute 'OPC.UA.DA' := '1'}
	P2143_RUN            AT %Q*   :BOOL;    //P2143 Run Command
	{attribute 'OPC.UA.DA' := '1'}
	P2142_RUN            AT %Q*   :BOOL;    //P2142 Run Command
	{attribute 'OPC.UA.DA' := '1'}
	P2145_RUN            AT %Q*   :BOOL;    //P2145 Run Command
	{attribute 'OPC.UA.DA' := '1'}
	P2150_RUN            AT %Q*   :BOOL;    //P2150 Run Command
	
	{attribute 'OPC.UA.DA' := '1'}
	P3085_RUN            AT %Q*   :BOOL;    //P3085 Run Command
	{attribute 'OPC.UA.DA' := '1'}
	P3090_RUN            AT %Q*   :BOOL;    //P3090 Run Command
	{attribute 'OPC.UA.DA' := '1'}
	P3095_RUN            AT %Q*   :BOOL;    //P3095 Run Command	
//---------------------------------Motor Feedback-------------------------------------------------
	{attribute 'OPC.UA.DA' := '1'}
	P2130_Faulted            AT %I*   :BOOL;    //P2130 Faulted 
	{attribute 'OPC.UA.DA' := '1'}
	P2135_Faulted            AT %I*   :BOOL;    //P2135 Faulted 
	{attribute 'OPC.UA.DA' := '1'}
	P2140_Faulted            AT %I*   :BOOL;    //P2140 Faulted 
	{attribute 'OPC.UA.DA' := '1'}
	P2143_Faulted            AT %I*   :BOOL;    //P2143 Faulted 
	{attribute 'OPC.UA.DA' := '1'}
	P2142_Faulted            AT %I*   :BOOL;    //P2142 Faulted 
	{attribute 'OPC.UA.DA' := '1'}
	P2145_Faulted            AT %I*   :BOOL;    //P2145 Faulted
 
	{attribute 'OPC.UA.DA' := '1'}
	P2150_Faulted            AT %I*   :BOOL;    //P2150 Faulted 
	{attribute 'OPC.UA.DA' := '1'}
	P3085_Faulted            AT %I*   :BOOL;    //P3085 Faulted 
	{attribute 'OPC.UA.DA' := '1'}
	P3090_Faulted            AT %I*   :BOOL;    //P3090 Faulted 
	{attribute 'OPC.UA.DA' := '1'}
	P3095_Faulted            AT %I*   :BOOL;    //P3095 Faulted 
//---------------------------------Disconnect Status------------------------------------------------- 
	{attribute 'OPC.UA.DA' := '1'}
	DS_P2130            AT %I*  :BOOL;  //P2130 Disconnect
	{attribute 'OPC.UA.DA' := '1'}
	DS_P2135            AT %I*  :BOOL;  //P2135 Disconnect
	{attribute 'OPC.UA.DA' := '1'}
	DS_P2140            AT %I*  :BOOL;  //P2140 Disconnect
	{attribute 'OPC.UA.DA' := '1'}
	DS_P2143            AT %I*  :BOOL;  //P2143 Disconnect
	{attribute 'OPC.UA.DA' := '1'}
	DS_P2141            AT %I*  :BOOL;  //P2141 Disconnect
	{attribute 'OPC.UA.DA' := '1'}
	DS_P2142            AT %I*  :BOOL;  //P2142 Disconnect
	{attribute 'OPC.UA.DA' := '1'}
	DS_P2145            AT %I*  :BOOL;  //P2145 Disconnect
	{attribute 'OPC.UA.DA' := '1'}
	DS_P2146            AT %I*  :BOOL;  //P2146 Disconnect
	{attribute 'OPC.UA.DA' := '1'}
	DS_P2150            AT %I*  :BOOL;  //P2150 Disconnect
	{attribute 'OPC.UA.DA' := '1'}
	DS_P3080            AT %I*  :BOOL;  //P3080 Disconnect
	{attribute 'OPC.UA.DA' := '1'}
	DS_P3085            AT %I*  :BOOL;  //P3085 Disconnect
	{attribute 'OPC.UA.DA' := '1'}
	DS_P3090            AT %I*  :BOOL;  //P3090 Disconnect
	{attribute 'OPC.UA.DA' := '1'}
	DS_P3095            AT %I*  :BOOL;  //P3095 Disconnect
//---------------------------------Solenoid Valves------------------------------------------------- 
	{attribute 'OPC.UA.DA' := '1'}
   GR2140_01_Extend        AT %Q*:    BOOL; // P2140 Solenoid Extend   
	{attribute 'OPC.UA.DA' := '1'}
   GR2140_02_Extend        AT %Q*:    BOOL; // P2140 Solenoid Extend
	{attribute 'OPC.UA.DA' := '1'}
   PI2140_01_Extend        AT %Q*:    BOOL; // P2140 Solenoid Extend
	{attribute 'OPC.UA.DA' := '1'}
   PI2140_01_Retract       AT %Q*:    BOOL; // P2140 Solenoid Retract
	{attribute 'OPC.UA.DA' := '1'}
   PL2140_01_Extend        AT %Q*:    BOOL; // P2140 Solenoid Extend
	{attribute 'OPC.UA.DA' := '1'}
   GR2150_01_Extend        AT %Q*:    BOOL; // P2150 Solenoid Extend
	{attribute 'OPC.UA.DA' := '1'}
   PI2150_01_Extend        AT %Q*:    BOOL; // P2150 Solenoid Extend
	{attribute 'OPC.UA.DA' := '1'}
   PU2150_01_Extend        AT %Q*:    BOOL; // P2150 Solenoid Extend
	{attribute 'OPC.UA.DA' := '1'}
   PU2150_02_Extend        AT %Q*:    BOOL; // P2150 Solenoid Extend
	{attribute 'OPC.UA.DA' := '1'}
   PU2150_03_Extend        AT %Q*:    BOOL; // P2150 Solenoid Extend
	{attribute 'OPC.UA.DA' := '1'}
   PU2150_04_Extend        AT %Q*:    BOOL; // P2150 Solenoid Extend
//---------------------------------Encoder------------------------------------------------- 
	{attribute 'OPC.UA.DA' := '1'}
	ENC_9031_Raw	AT %I*:	UINT;	// Raw Encoder Value
	{attribute 'OPC.UA.DA' := '1'}
	ENC_9031_OK			: BOOL;
	{attribute 'OPC.UA.DA' := '1'}
	ENC_9031_Period	AT %I*:	UDINT;	// Encoder Period, channel 1, 100ns resolution
	
	{attribute 'OPC.UA.DA' := '1'}
	ENC_9091_Raw	AT %I*:	UINT;	// Raw Encoder Value
	{attribute 'OPC.UA.DA' := '1'}
	ENC_9091_OK			: BOOL;
	{attribute 'OPC.UA.DA' := '1'}
	ENC_9091_Period	AT %I*:	UDINT;	// Encoder Period, channel 1, 100ns resolution
	
	Sorter_P2140Name				: STRING[5];
	Sorter_P2150Name				: STRING[5];
//---------------------------------WcStates-------------------------------------------------
	{attribute 'OPC.UA.DA' := '1'}
 	RIO1151_WcState AT %I*				: BOOL;		// Remote IO Block 1151
	{attribute 'OPC.UA.DA' := '1'}
	RIO2151_WcState AT %I*				: BOOL;		// Remote IO Block 2151
	{attribute 'OPC.UA.DA' := '1'}
	RIO3171_WcState AT %I*				: BOOL;		// Remote IO Block 3171
	{attribute 'OPC.UA.DA' := '1'}
	RIO4141_WcState AT %I*				: BOOL;		// Remote IO Block 4141
	{attribute 'OPC.UA.DA' := '1'}
	RIO7151_WcState AT %I*				: BOOL;		// Remote IO Block 7151
	{attribute 'OPC.UA.DA' := '1'}
	RIO8171_WcState AT %I*				: BOOL;		// Remote IO Block 8171
	{attribute 'OPC.UA.DA' := '1'}
	RIO9191_WcState AT %I*				: BOOL;		// Remote IO Block 9191
	{attribute 'OPC.UA.DA' := '1'}
	{attribute 'OPC.UA.DA' := '1'}
	RIO10161_WcState AT %I*				: BOOL;		// Remote IO Block 10161
	{attribute 'OPC.UA.DA' := '1'}
	RIO11171_WcState AT %I*				: BOOL;		// Remote IO Block 11171
	{attribute 'OPC.UA.DA' := '1'}
	RIO12182_WcState AT %I*				: BOOL;		// Remote IO Block 12812
	{attribute 'OPC.UA.DA' := '1'}

	{attribute 'OPC.UA.DA' := '1'}
	EthernetAdapter_State AT %I*	    : UINT;		// Ethernet Adapter State
 //---------------------------------EAP-------------------------------------------------
//Published
  To205_P2130_IsRunning	AT %Q*:	BOOL; 
  To205_P3095_SendingProduct AT %Q*: BOOL; 
//Subscribed
  From205_P3100_IsRunning AT %I*: BOOL;
  From205_P2125_SendingProduct AT %I*: BOOL;


END_VAR

// ---- GVLs/GVL_Logging.TcGVL
// Comment out attribute to allow direct access to this variable
// {attribute 'qualified_only'} 
VAR_GLOBAL PERSISTENT
	nMessageLogEnable:				UDINT;		// 32 separate log events to enable
	nBarcodeLogEnable:				UDINT;		// 32 separate log events to enable
	nServerLogEnable:				UDINT;		// 32 separate log events to enable, default to enabled, turn off 
	nItemBufferLogEnable:			UDINT;		// 32 separate log events to enable	
	nItemBufferLogEnableP2140:		UDINT;		// 32 separate log events to enable	
	nItemBufferLogEnableP2150:		UDINT;		// 32 separate log events to enable	
	nSorterLogEnable:				UDINT;		// 32 separate log events to enable	
	nSorterLogEnableP2140:			UDINT;		// 32 separate log events to enable	
	nSorterLogEnableP2150:			UDINT;		// 32 separate log events to enable	
	nDivertLogEnable:				UDINT;		// 32 separate log events to enable	
	nDivertLogEnableP2140:			UDINT;		// 32 separate log events to enable	
	nDivertLogEnableP2150:			UDINT;		// 32 separate log events to enable	
	nSortBufferLogEnable:			UDINT;		// 32 separate log events to enable	
	nSortBufferLogEnableP2140:		UDINT;		// 32 separate log events to enable	
	nSortBufferLogEnableP2150:		UDINT;		// 32 separate log events to enable	
END_VAR

VAR_GLOBAL CONSTANT
	// To enable a specific log, turn ON the bit associate with that log type in the Enable UDINT 
	// The constants below correspond to the bit number within the UDINT

	// Use E_MessageIds as constants for message logging
	// Barcode Logging
	TRIGGER_PE		:	INT := 0;
	TRIGGER			:	INT := 1;
	BCR_S2140_01_LOG	:	INT := 2;
	BCR_S2141_01_LOG	:	INT := 3;
	BCR_S2150_01_LOG	:	INT := 4;
	BCR_S3080_01_LOG	:	INT := 5;

	// Barcode Logging
	BUFFER_LOG	:	INT := 0;	
	// Item Buffer Logging
	ARRIVALS		:	INT := 0;
	TRANSPORT		: 	INT := 1;
	UPDATE			: 	INT := 2;
	// nDivertLogEnable constants
	// Increase for additional Diverts
	DIVERT_DECISION	:	INT := 0;
	DIVERT1			:	INT := 1;
	DIVERT2			:	INT := 2;
	DIVERT3			:	INT := 3;
	DIVERT4			:	INT := 4;
	DIVERT5			:	INT := 5;
	DIVERT6			:	INT := 6;
	DIVERT7			:	INT := 7;
	DIVERT8			:	INT := 8;
	CONFIRM1		:	INT := 16;
	CONFIRM2		:	INT := 17;
	CONFIRM3		:	INT := 18;
	CONFIRM4		:	INT := 19;
	CONFIRM5		:	INT := 20;
	CONFIRM6		:	INT := 21;
	CONFIRM7		:	INT := 22;
	CONFIRM8		:	INT := 23;
	LANEFULL		:	INT := 31;
	// nSorterLogEnable constants
	SORTER_INDUCT		:	INT	:= 0;
	SORTER_INDUCT_PE	:	INT	:= 1;
	SORTER_DIVERTS		:	INT	:= 2;
	SORTER_CONFIRMS		:	INT	:= 3;
	SORTER_DUMP			:	INT	:= 4;
	SORTER_TEMPID		:	INT	:= 5;
	SORTER_HEIGHT_PE	:	INT := 6;
	SORTER_DISCHARGE_PE	:	INT	:= 7;
	SORTER_DESTINATION_LU	:	INT	:= 8;
	// Sorter buffer constants
	BUFFER_ARRIVAL			:	INT := 0;
	BUFFER_MISSINDUCT		: 	INT := 1;
	BUFFER_TEMPINDUCT		:	INT := 2;
	BUFFER_INDUCT			:	INT := 3;
	BUFFER_LATEINDUCT		:	INT := 4;
	BUFFER_REPLACEINDUCT	:	INT := 5;
	BUFFER_UPDATEINDUCT		:	INT := 6;
	BUFFER_UPDATEDEST		:	INT := 7;
	BUFFER_DUMP				:	INT := 8;
	BUFFER_UNASSIGNED		:	INT := 9;
	BUFFER_DESTINDEX		:	INT := 10;
END_VAR

// ---- GVLs/GVL_SorterItems.TcGVL
//{attribute 'qualified_only'}
VAR_GLOBAL
	// Default Destination per Sorter/divert
	P2140_DefaultDestination:		DINT;	// Input default destination update from Host messaging(MsgControl.RECEIVE)
	P2150_DefaultDestination:		DINT;	// Input default destination update from Host messaging(MsgControl.RECEIVE)

	st_SorterArrivalBuffer_P2140:		ST_ItemBuffer;		// Output from the Barcode Reader to the sorter
	st_ArrivalFdbkIn_P2140: 			ST_ItemBufferFdbk;
	st_ArrivalFdbkOut_P2140:			ST_ItemBufferFdbk;

	st_SorterArrivalBuffer_P2150:		ST_ItemBuffer;		// Output from the Barcode Reader to the sorter
	st_ArrivalFdbkIn_P2150:				ST_ItemBufferFdbk;
	st_ArrivalFdbkOut_P2150:			ST_ItemBufferFdbk;
	
	st_SorterTransportBuffer_P2140:		ST_ItemBuffer;		// Routing from the ARUP Host to the sorter
	st_TransportFdbkIn_P2140: 			ST_ItemBufferFdbk;
	st_TransportFdbkOut_P2140: 			ST_ItemBufferFdbk;

	st_SorterTransportBuffer_P2150:		ST_ItemBuffer;		// Routing from the ARUP Host to the sorter
	st_TransportFdbkIn_P2150: 			ST_ItemBufferFdbk;
	st_TransportFdbkOut_P2150: 			ST_ItemBufferFdbk;

	st_SorterUpdateBuffer:				ST_ItemBuffer;  	// Output from the sorter to update the host messaging (MsgControl)
	st_UpdateFdbkIn:					ST_ItemBufferFdbk;
	st_UpdateFdbkOut:					ST_ItemBufferFdbk;

	BlankItem					: ST_Item := (ID := '', UniqueID := 0
													, Destination := 0
													, DestinationIdx := 0
													, Status := E_StatusCode.No_Status
													, ExtStatus := E_StatusCode.No_Status
													, DeviceID := ''
													, MessageType := E_MessageIds.NoMessage_00);

END_VAR

// ---- POUs/MAIN.TcPOU
PROGRAM MAIN
VAR
	// Data persistence configuration
	rStartPersistentSave 		: R_TRIG; // Rising edge trigger to start persistent data save
	fbWritePersistentData 		: WritePersistentData;
	tonPersistentSave	:	TON := (PT := T#1M);
	tpBroadcastSave		:	TP	:= (PT := T#100MS);
	PLCPersistentSave			AT %Q*	: BOOL;
	ADSPort						:	UINT := 0;
	In_ResetAllMetrics			: 	BOOL;
END_VAR
VAR PERSISTENT
	EAP_205 : ST_EAP_DEVICE ;	
END_VAR

SystemSafety();
BarCodeReaders();
CommStatus();
Solenoids();
Conveyors();
Sorter();
Log_Diverts_P2140();
Log_Diverts_P2150();
Photoeyes();
ProxSensors();
ServerControl();
Singulation_Control();
System();
P_PulseCountDist();
GVL_IO.INIT := FALSE;


// Reset when Timer is Done
tonPersistentSave(IN := NOT tpBroadcastSave.Q);

// Catch the .Q of the persistent save timer to trigger a save pulse
tpBroadcastSave(IN := tonPersistentSave.Q);
// Set the Persistent save outputs to the .Q of the pulse
PLCPersistentSave := tpBroadcastSave.Q;

// Check for persistent item save
//rStartPersistentSave(CLK := tpBroadcastSave.Q);
// Execute a Persistent save here
// System PORT is 851
fbWritePersistentData(netid:= '', PORT:=851, Start:=tonPersistentSave.Q, tmout:=T#1S);

// Convert HMI EAP IP Address(es) to correct format
MEMCPY(destAddr    := ADR(EAP_205.Publisher.HMI_IPAddrDisp),srcaddr :=ADR(EAP_205.Publisher.IPAddr), n := 4);
IF ((EAP_205.Publisher.HMI_IPAddrDisp[0] <> EAP_205.Publisher.HMI_IPAddr[0]) AND EAP_205.Publisher.HMI_IPAddr[0] > 0)
   OR ((EAP_205.Publisher.HMI_IPAddrDisp[1] <> EAP_205.Publisher.HMI_IPAddr[1]) AND EAP_205.Publisher.HMI_IPAddr[1] > 0)
   OR ((EAP_205.Publisher.HMI_IPAddrDisp[2] <> EAP_205.Publisher.HMI_IPAddr[2]) AND EAP_205.Publisher.HMI_IPAddr[2] > 0)
   OR ((EAP_205.Publisher.HMI_IPAddrDisp[3] <> EAP_205.Publisher.HMI_IPAddr[3]) AND EAP_205.Publisher.HMI_IPAddr[3] > 0)
   THEN
    MEMCPY(destAddr    := ADR(EAP_205.Publisher.IPAddr),srcaddr :=ADR(EAP_205.Publisher.HMI_IPAddr), n := 4);
END_IF

END_PROGRAM

// ---- POUs/SystemSafety.TcPOU
PROGRAM SystemSafety
VAR
	{attribute 'OPC.UA.DA' := '1'}
	System_SafetyState : ST_SafetyState;
	{attribute 'OPC.UA.DA' := '1'}

	{attribute 'OPC.UA.DA' := '1'}
	Safety_SystemEstopsOK AT %I* : BOOL;
	{attribute 'OPC.UA.DA' := '1'}
	Safety_PanelEstop AT %I* : BOOL;
END_VAR

// Set System Safety Variables 
System_SafetyState.ErrAck := System.Safety_Reset;
System_SafetyState.CommErrAck := System.Safety_Reset;
System_SafetyState.Reset := System.Safety_Reset;
System_SafetyState.Run := TRUE;

END_PROGRAM

// ---- POUs/System.TcPOU
PROGRAM System
VAR
	{attribute 'OPC.UA.DA' := '0'}
	SysStateCntrlSts        	:    ST_EquipmentStatus;    // System State/Control/Status Data
    SysState                	:    FB_SystemCntrl;
    SysStateCntrl_StatePB       :    ST_StateCntrlPB;

    SysIntlksAllOk AT %Q*    	:    BOOL;    // Bit to show that System interlocks are OK   
    SysEventsAllOk AT %Q*		: 	BOOL;    // Bit to show that Syetem events are all OK If system events are needed use event manager FB tie to here
	
	ConvDefaultState AT %Q*		: 	E_StateCntrl := E_StateCntrl.stManual;	// The default state of all conveyors
	Sys_SimActive AT %Q*		: 	BOOL;	// Bit for simulation
	
	{attribute 'OPC.UA.DA' := '1'}
	HMI_PBSysStart:	BOOL;
	{attribute 'OPC.UA.DA' := '1'}
	HMI_PBSysStop:	BOOL;
	{attribute 'OPC.UA.DA' := '1'}
	HMI_PBSysReset:	BOOL;
	
	SysShrtPulseTmr: FB_Flasher;
	SysShrtPlsOnTime: TIME := T#750MS;
	SysShrtPlsOffTime: TIME := T#750MS;
	
	Cnvyr_Auto AT %Q*:	BOOL;		// Bit to send to all conveyors to put them in Auto mode
	Cnvyr_Manual AT %Q*:	BOOL;	// Bit to send to all conveyors to put them in Manual mode
	Cnvyr_Offline AT %Q*:	BOOL;	// Bit to send to all conveyors to put them in Offline mode -- Not used here
	Cnvyr_Reset AT %Q*:	BOOL;		// Bit to send to all conveyors to reset faults, safeties and etc
	Safety_Reset:	BOOL;
	tpSafetyReset:		TP := (PT := T#250MS);
	fSafetyReset:		F_TRIG;

	tpConvReset:		TP := (PT := T#250MS);
	
	Cnvyr_AlertTime:	TIME := T#5S;	
	Cnvyr_DelayTime:	TIME := T#1S;	
	Start_PulseWidth:	TIME := T#100MS;
	AlertDelay: FB_AlrtStrtDelay;
	
	nStatusArrayIndex : DINT;	// Increment to process the SysEquipStatusArray
	nTempStsIndex : DINT := 0;	// Used to Prevent Status Array Index duplicate assignments 

	ConveyorHasWarn: BOOL;
	ConveyorHasFault: BOOL;
	ConveyorIsSleeping: BOOL;
	ConveyorInAuto: BOOL;
	nTempRemoteIndex: DINT := 0;	//Temporary Remote Index to Simplify Code
	
END_VAR

VAR PERSISTENT    {attribute 'OPC.UA.DA' := '1'}
    cfgSysStateIntlksArry: ARRAY [0..15] OF ST_CfgEvents;
    {attribute 'OPC.UA.DA' := '1'}
    cfgSysStateEvntsArry: ARRAY [0..15] OF ST_CfgEvents;
END_VAR

tpConvReset.PT := T#3S;

// Send out reset PB put here in case added logic was needed
SysStateCntrl_StatePB.ResetPB := GVL_IO.PB_SysReset OR HMI_PBSysReset OR GVL_IO.PB_RemoteReset_3211 OR GVL_IO.PB_RemoteReset_8251 OR GVL_IO.PB_RemoteReset_10221;
SysStateCntrl_StatePB.AutoPB := (HMI_PBSysStart OR GVL_IO.PB_SysStart) AND SysIntlksAllOk;
SysStateCntrl_StatePB.StopPB := HMI_PBSysStop OR (NOT GVL_IO.PB_SysStop);

// Set up system short pulse for alarm beacons, horns ets
SysShrtPulseTmr(In_Trig:= TRUE , Cfg_OnTime:= SysShrtPlsOnTime, Cfg_OffTime:= SysShrtPlsOffTime, Output=> );

// Set up System Interlocks

SysState.In_SystemIntlks.0 := GVL_IO.SystemAirPressure;
SysState.In_SystemIntlks.1 := SystemSafety.System_SafetyState.InRun;

(*
// Setup the InterlockArray since persistent data items cannot by initilaized the same
// Index 0
cfgSysStateIntlksArry[0].Description := 'System Air Pressure';
cfgSysStateIntlksArry[0].DeviceLabel := 'System';
cfgSysStateIntlksArry[0].OKState := TRUE;
// Index 1
cfgSysStateIntlksArry[1].Description := 'Safety in Run';
cfgSysStateIntlksArry[1].DeviceLabel := 'Safety';
cfgSysStateIntlksArry[1].OKState := TRUE;
*)

// Set up System Events

SysState.In_SystemEvents.0 := SystemSafety.Safety_PanelEstop;
SysState.In_SystemEvents.1 := GVL_IO.Remote_PullCord2142_OK;
SysState.In_SystemEvents.2 := GVL_IO.Remote_PullCord2150_OK;
SysState.In_SystemEvents.3 := SystemSafety.System_SafetyState.ComErr;
SysState.In_SystemEvents.4 := SystemSafety.System_SafetyState.FBErr;
SysState.In_SystemEvents.5 := SystemSafety.System_SafetyState.OtherErr;

(*
// Setup the EventArray since persistent data items cannot by initilaized the same
// Index 0
cfgSysStateEvntsArry[0].Description := 'Panel E-Stop';
cfgSysStateEvntsArry[0].DeviceLabel := 'PB1';
cfgSysStateEvntsArry[0].OKState := TRUE;
cfgSysStateEvntsArry[0].StopCode := E_StopCodes.SystemStop;
// Index 1
cfgSysStateEvntsArry[1].Description := 'P2142 Pull cord OK';
cfgSysStateEvntsArry[1].DeviceLabel := 'P2142';
cfgSysStateEvntsArry[1].OKState := TRUE;
cfgSysStateEvntsArry[1].StopCode := E_StopCodes.SystemStop;
// Index 2
cfgSysStateEvntsArry[2].Description := 'P2150 Pull cord OK';
cfgSysStateEvntsArry[2].DeviceLabel := 'P2150';
cfgSysStateEvntsArry[2].OKState := TRUE;
cfgSysStateEvntsArry[2].StopCode := E_StopCodes.SystemStop;
// Index 3
cfgSysStateEvntsArry[3].Description := 'Safety Comm Error';
cfgSysStateEvntsArry[3].DeviceLabel := 'SYSTEM';
cfgSysStateEvntsArry[3].OKState := FALSE;
cfgSysStateEvntsArry[3].StopCode := E_StopCodes.SystemStop;
// Index 4
cfgSysStateEvntsArry[4].Description := 'Safety FunctionBlock Error';
cfgSysStateEvntsArry[4].DeviceLabel := 'SYSTEM';
cfgSysStateEvntsArry[4].OKState := FALSE;
cfgSysStateEvntsArry[4].StopCode := E_StopCodes.SystemStop;
// Index 5
cfgSysStateEvntsArry[5].Description := 'Safety Error';
cfgSysStateEvntsArry[5].DeviceLabel := 'SYSTEM';
cfgSysStateEvntsArry[5].OKState := FALSE;
cfgSysStateEvntsArry[5].StopCode := E_StopCodes.SystemStop;
*)
// Function Call
SysState(
    In_p_EquipStatePB:= SysStateCntrl_StatePB,
	Cfg_EquipLabel := 'Building 1.5',  
    Cfg_EquipIntlksArry:= cfgSysStateIntlksArry,
    Cfg_EquipEvntsArry:= cfgSysStateEvntsArry, 
    Sts_EquipState := SysStateCntrlSts,
	Out_Reset => 
);

SysIntlksAllOk := SysState.Sts_All_Intlks_OK;
SysEventsAllOk := SysState.Sts_All_Evnts_OK;

// Separate Standard/safety resets
tpSafetyReset(IN:= SysState.Out_Reset);
// On While the timer is timing
Safety_Reset := tpSafetyReset.Q;

// On when the safety pulse goes low
fSafetyReset(CLK := tpSafetyReset.Q);
tpConvReset(IN := fSafetyReset.Q);
// On while the timer is timing
Cnvyr_Reset := tpConvReset.Q;

// Set up Start up delay and Auto/Manual control for conveyors

// Offline is set up in conveyors but has no logic here controlling it(This could be added here)
AlertDelay(
	In_StrtPulse:= SysState.Out_Auto , 
	In_StpPulse:= SysState.Out_Stop,
	CFG_AlertTime:= Cnvyr_AlertTime, 
	CFG_WaitTime:= Cnvyr_DelayTime,
	CFG_PulseTime:= Start_PulseWidth,
	In_ManTstTrig:= , 
	In_BypssDelay:= , 
	Out_Timed => Cnvyr_Auto,
	Out_Pulse => , 
	Out_Alert=> GVL_IO.HornMainPanel, 
	WaitActive=> );

Cnvyr_Manual:= SysState.Out_Stop; 	

//===========================================================================================
// Serialize the reporting equipment

// Set the value of System_Equip_Count, TempStsIndex should always match the number of identified statuses
GVL_EquipArrays.nSystemEquip_Count := nTempStsIndex;

// Control tower light
// Initialize the Equipment state detection
ConveyorHasWarn := 0;
ConveyorHasFault := 0;
ConveyorIsSleeping := 0;
ConveyorInAuto := 0;

//Conveyor Equipment
// Adjust GVL_EquipArrays.cEQUIP_COUNT_MAX to accommodate all of the equipment to monitor
IF GVL_EquipArrays.nEquipIndex <> 0 THEN
    FOR nStatusArrayIndex := 1 TO GVL_EquipArrays.nEquipIndex BY 1 DO
		IF nStatusArrayIndex <= GVL_EquipArrays.cEQUIP_COUNT_MAX THEN
			// Test for an already assigned Index value, but only to the outbound index, eventually this will populate the inbound value
			IF GVL_EquipArrays.aEquipStatusArray_Out[nStatusArrayIndex].RemIndex = 0 THEN
				// Increment the TempStsIndex only when we need to
				nTempStsIndex := nTempStsIndex + 1;
				// Assign the Remote Index to the Conveyor Status Data Item
				GVL_EquipArrays.aEquipStatusArray_Out[nStatusArrayIndex].RemIndex := nTempStsIndex;
			END_IF
			// Assign the Conveyor Status Value to the Status Array
			nTempRemoteIndex := GVL_EquipArrays.aEquipStatusArray_Out[nStatusArrayIndex].RemIndex;
			GVL_EquipArrays.aSystemEquipStatusArray[nTempRemoteIndex] := GVL_EquipArrays.aEquipStatusArray_In[nStatusArrayIndex];
		END_IF
    END_FOR
END_IF

